C07261=1094.905,99.081,438.619,176.128,17.125,152.423
C07262=1094.899,98.832,438.636,176.125,17.124,152.424
C07263=1094.893,98.582,438.654,176.123,17.123,152.424
C07264=1094.888,98.333,438.673,176.120,17.123,152.424
C07265=1094.882,98.083,438.691,176.117,17.121,152.425
C07266=1094.877,97.834,438.709,176.115,17.121,152.425
C07267=1094.870,97.585,438.726,176.112,17.120,152.425
C07268=1094.865,97.336,438.745,176.110,17.119,152.426
C07269=1094.859,97.086,438.763,176.108,17.118,152.426
C07270=1094.854,96.837,438.781,176.106,17.117,152.426
C07271=1094.848,96.587,438.799,176.103,17.117,152.426
C07272=1094.843,96.339,438.818,176.100,17.115,152.427
C07273=1094.836,96.063,438.837,176.098,17.115,152.427
C07274=1094.830,95.788,438.857,176.095,17.114,152.427
C07275=1094.824,95.513,438.877,176.093,17.113,152.428
C07276=1094.817,95.237,438.896,176.090,17.112,152.428
C07277=1094.812,94.988,438.915,176.087,17.111,152.428
C07278=1094.806,94.739,438.933,176.085,17.110,152.429
C07279=1094.801,94.490,438.951,176.082,17.109,152.429
C07280=1094.794,94.240,438.969,176.080,17.108,152.429
C07281=1094.790,93.991,438.987,176.077,17.108,152.430
C07282=1094.784,93.741,439.005,176.075,17.107,152.430
C07283=1094.778,93.492,439.022,176.073,17.106,152.430
C07284=1094.772,93.243,439.040,176.070,17.104,152.430
C07285=1094.767,92.993,439.059,176.068,17.104,152.431
C07286=1094.761,92.744,439.077,176.065,17.103,152.431
C07287=1094.756,92.495,439.094,176.063,17.102,152.431
C07288=1094.750,92.245,439.112,176.061,17.101,152.432
C07289=1094.744,91.996,439.130,176.059,17.101,152.432
C07290=1094.739,91.747,439.148,176.056,17.099,152.432
C07291=1094.733,91.497,439.166,176.054,17.099,152.432
C07292=1094.728,91.248,439.184,176.051,17.097,152.433
C07293=1094.722,90.999,439.201,176.048,17.097,152.433
C07294=1094.716,90.749,439.219,176.046,17.096,152.433
C07295=1094.711,90.500,439.237,176.044,17.095,152.434
C07296=1094.705,90.251,439.254,176.042,17.094,152.434
C07297=1094.699,90.002,439.272,176.039,17.093,152.434
C07298=1094.693,89.753,439.290,176.037,17.093,152.434
C07299=1094.688,89.504,439.307,176.034,17.092,152.435
C07300=1094.682,89.254,439.325,176.032,17.091,152.435
C07301=1094.676,89.005,439.343,176.030,17.090,152.435
C07302=1094.670,88.755,439.361,176.027,17.088,152.436
C07303=1094.665,88.506,439.378,176.025,17.088,152.436
C07304=1094.659,88.257,439.396,176.022,17.087,152.436
C07305=1094.653,88.007,439.414,176.020,17.086,152.436
C07306=1094.647,87.758,439.431,176.017,17.085,152.437
C07307=1094.642,87.509,439.449,176.015,17.084,152.437
C07308=1094.636,87.260,439.466,176.013,17.083,152.437
C07309=1094.631,87.010,439.484,176.011,17.083,152.437
C07310=1094.625,86.761,439.501,176.008,17.081,152.438
C07311=1094.620,86.512,439.519,176.006,17.081,152.438
C07312=1094.613,86.262,439.537,176.004,17.079,152.438
C07313=1094.608,86.013,439.554,176.001,17.078,152.439
C07314=1094.602,85.764,439.572,175.999,17.078,152.439
C07315=1094.596,85.514,439.590,175.996,17.076,152.439
C07316=1094.591,85.264,439.607,175.994,17.076,152.439
C07317=1094.586,85.015,439.624,175.992,17.074,152.440
C07318=1094.580,84.766,439.642,175.990,17.074,152.440
C07319=1094.574,84.517,439.660,175.987,17.073,152.440
C07320=1094.568,84.268,439.677,175.985,17.072,152.440
C07321=1094.563,84.018,439.694,175.982,17.071,152.441
C07322=1094.558,83.769,439.712,175.981,17.070,152.441
C07323=1094.552,83.519,439.730,175.978,17.069,152.441
C07324=1094.546,83.270,439.747,175.976,17.068,152.441
C07325=1094.540,83.021,439.763,175.973,17.067,152.442
C07326=1094.535,82.772,439.781,175.970,17.066,152.442
C07327=1094.529,82.523,439.799,175.969,17.065,152.442
C07328=1094.523,82.273,439.817,175.966,17.064,152.442
C07329=1094.518,82.023,439.833,175.964,17.063,152.443
C07330=1094.512,81.774,439.851,175.961,17.062,152.443
C07331=1094.507,81.525,439.869,175.959,17.061,152.443
C07332=1094.501,81.276,439.885,175.957,17.060,152.443
C07333=1094.495,81.026,439.903,175.955,17.059,152.444
C07334=1094.489,80.777,439.920,175.952,17.058,152.444
C07335=1094.484,80.527,439.937,175.950,17.058,152.444
C07336=1094.478,80.278,439.955,175.947,17.056,152.445
C07337=1094.472,80.003,439.974,175.945,17.055,152.445
C07338=1094.466,79.728,439.993,175.943,17.054,152.445
C07339=1094.460,79.452,440.012,175.940,17.053,152.445
C07340=1094.454,79.177,440.031,175.937,17.052,152.446
C07341=1094.448,78.928,440.049,175.935,17.050,152.446
C07342=1094.443,78.678,440.066,175.933,17.050,152.446
C07343=1094.437,78.429,440.082,175.930,17.048,152.446
C07344=1094.431,78.180,440.100,175.928,17.048,152.447
C07345=1094.425,77.930,440.117,175.926,17.047,152.447
C07346=1094.420,77.681,440.135,175.924,17.046,152.447
C07347=1094.414,77.431,440.151,175.921,17.045,152.447
C07348=1094.408,77.182,440.169,175.919,17.044,152.448
C07349=1094.403,76.933,440.186,175.917,17.043,152.448
C07350=1094.397,76.684,440.202,175.915,17.042,152.448
C07351=1094.391,76.434,440.220,175.912,17.040,152.448
C07352=1094.385,76.185,440.237,175.910,17.040,152.448
C07353=1094.379,75.935,440.254,175.908,17.039,152.449
C07354=1094.374,75.686,440.271,175.906,17.038,152.449
C07355=1094.369,75.437,440.288,175.903,17.037,152.449
C07356=1094.363,75.188,440.305,175.901,17.036,152.450
C07357=1094.357,74.938,440.322,175.899,17.034,152.450
C07358=1094.352,74.689,440.339,175.897,17.034,152.450
C07359=1094.345,74.439,440.356,175.894,17.033,152.450
C07360=1094.340,74.190,440.374,175.892,17.032,152.450
C07361=1094.334,73.940,440.390,175.889,17.031,152.451
C07362=1094.329,73.691,440.407,175.888,17.030,152.451
C07363=1094.323,73.442,440.424,175.885,17.028,152.451
C07364=1094.318,73.192,440.441,175.883,17.028,152.451
C07365=1094.312,72.944,440.458,175.880,17.026,152.452
C07366=1094.306,72.694,440.475,175.879,17.026,152.452
C07367=1094.300,72.445,440.491,175.876,17.024,152.452
C07368=1094.295,72.196,440.509,175.874,17.023,152.452
C07369=1094.290,71.946,440.526,175.872,17.022,152.452
C07370=1094.283,71.696,440.542,175.870,17.022,152.453
C07371=1094.278,71.447,440.560,175.867,17.020,152.453
C07372=1094.272,71.197,440.576,175.865,17.019,152.453
C07373=1094.266,70.948,440.593,175.863,17.018,152.453
C07374=1094.261,70.699,440.610,175.861,17.017,152.453
C07375=1094.255,70.449,440.627,175.858,17.016,152.454
C07376=1094.250,70.200,440.644,175.856,17.015,152.454
C07377=1094.243,69.951,440.660,175.854,17.014,152.454
C07378=1094.238,69.701,440.677,175.852,17.013,152.454
C07379=1094.232,69.452,440.694,175.849,17.011,152.455
C07380=1094.227,69.202,440.710,175.847,17.011,152.455
C07381=1094.221,68.954,440.727,175.845,17.010,152.455
C07382=1094.216,68.704,440.744,175.843,17.008,152.455
C07383=1094.210,68.455,440.761,175.840,17.007,152.456
C07384=1094.204,68.205,440.777,175.838,17.007,152.456
C07385=1094.198,67.956,440.794,175.836,17.005,152.456
C07386=1094.193,67.707,440.811,175.834,17.004,152.456
C07387=1094.187,67.457,440.827,175.831,17.003,152.456
C07388=1094.182,67.208,440.844,175.830,17.002,152.457
C07389=1094.176,66.958,440.861,175.827,17.001,152.457
C07390=1094.170,66.709,440.877,175.825,17.000,152.457
C07391=1094.164,66.460,440.894,175.824,16.999,152.457
C07392=1094.158,66.211,440.911,175.821,16.998,152.457
C07393=1094.153,65.961,440.928,175.819,16.997,152.458
C07394=1094.147,65.711,440.944,175.817,16.995,152.458
C07395=1094.141,65.462,440.960,175.815,16.995,152.458
C07396=1094.136,65.212,440.977,175.812,16.993,152.458
C07397=1094.130,64.963,440.993,175.810,16.992,152.458
C07398=1094.125,64.714,441.011,175.808,16.991,152.459
C07399=1094.119,64.465,441.027,175.806,16.990,152.459
C07400=1094.113,64.215,441.043,175.803,16.989,152.459
C07401=1094.106,63.940,441.061,175.801,16.988,152.459
C07402=1094.100,63.664,441.079,175.799,16.987,152.460
C07403=1094.093,63.389,441.097,175.796,16.986,152.460
C07404=1094.087,63.113,441.115,175.794,16.984,152.460
C07405=1094.082,62.864,441.133,175.792,16.983,152.460
C07406=1094.076,62.615,441.149,175.789,16.982,152.461
C07407=1094.070,62.366,441.165,175.787,16.981,152.461
C07408=1094.064,62.116,441.182,175.785,16.980,152.461
C07409=1094.058,61.867,441.198,175.783,16.979,152.461
C07410=1094.053,61.617,441.215,175.781,16.978,152.461
C07411=1094.047,61.368,441.231,175.778,16.977,152.462
C07412=1094.041,61.119,441.247,175.777,16.976,152.462
C07413=1094.035,60.869,441.264,175.774,16.974,152.462
C07414=1094.029,60.620,441.280,175.772,16.974,152.462
C07415=1094.024,60.370,441.297,175.770,16.972,152.462
C07416=1094.018,60.121,441.313,175.768,16.971,152.463
C07417=1094.012,59.871,441.328,175.765,16.970,152.463
C07418=1094.006,59.622,441.345,175.763,16.969,152.463
C07419=1094.000,59.372,441.361,175.762,16.968,152.463
C07420=1093.995,59.123,441.378,175.759,16.967,152.463
C07421=1093.989,58.873,441.394,175.757,16.966,152.464
C07422=1093.983,58.624,441.410,175.755,16.964,152.464
C07423=1093.978,58.375,441.426,175.753,16.964,152.464
C07424=1093.972,58.126,441.442,175.750,16.962,152.464
C07425=1093.966,57.877,441.459,175.749,16.961,152.464
C07426=1093.960,57.627,441.475,175.746,16.960,152.464
C07427=1093.955,57.377,441.491,175.744,16.959,152.465
C07428=1093.949,57.128,441.507,175.742,16.958,152.465
C07429=1093.943,56.878,441.524,175.740,16.957,152.465
C07430=1093.937,56.629,441.540,175.738,16.956,152.465
C07431=1093.931,56.380,441.556,175.736,16.954,152.465
C07432=1093.926,56.131,441.572,175.734,16.954,152.466
C07433=1093.920,55.881,441.588,175.731,16.952,152.466
C07434=1093.915,55.631,441.604,175.729,16.951,152.466
C07435=1093.909,55.382,441.621,175.727,16.949,152.466
C07436=1093.903,55.133,441.637,175.725,16.949,152.466
C07437=1093.897,54.883,441.653,175.723,16.947,152.467
C07438=1093.892,54.633,441.669,175.721,16.946,152.467
C07439=1093.886,54.385,441.685,175.719,16.945,152.467
C07440=1093.880,54.135,441.701,175.717,16.944,152.467
C07441=1093.874,53.886,441.717,175.715,16.943,152.467
C07442=1093.869,53.636,441.733,175.712,16.941,152.467
C07443=1093.863,53.387,441.749,175.710,16.941,152.468
C07444=1093.857,53.137,441.766,175.708,16.939,152.468
C07445=1093.852,52.888,441.781,175.706,16.938,152.468
C07446=1093.846,52.638,441.797,175.704,16.937,152.468
C07447=1093.841,52.389,441.813,175.702,16.935,152.468
C07448=1093.835,52.139,441.829,175.700,16.935,152.468
C07449=1093.829,51.890,441.845,175.698,16.933,152.469
C07450=1093.824,51.641,441.861,175.696,16.932,152.469
C07451=1093.818,51.391,441.877,175.693,16.931,152.469
C07452=1093.812,51.142,441.893,175.692,16.930,152.469
C07453=1093.806,50.892,441.909,175.690,16.929,152.469
C07454=1093.801,50.643,441.924,175.687,16.927,152.469
C07455=1093.795,50.394,441.941,175.686,16.926,152.470
C07456=1093.789,50.144,441.957,175.683,16.925,152.470
C07457=1093.783,49.894,441.972,175.681,16.924,152.470
C07458=1093.778,49.646,441.988,175.679,16.922,152.470
C07459=1093.772,49.396,442.004,175.677,16.921,152.470
C07460=1093.766,49.147,442.020,175.676,16.920,152.470
C07461=1093.761,48.897,442.036,175.673,16.919,152.471
C07462=1093.755,48.648,442.052,175.671,16.918,152.471
C07463=1093.750,48.399,442.068,175.669,16.916,152.471
C07464=1093.744,48.149,442.083,175.667,16.915,152.471
C07465=1093.738,47.873,442.101,175.664,16.914,152.471
C07466=1093.732,47.598,442.118,175.663,16.913,152.471
C07467=1093.726,47.321,442.136,175.660,16.911,152.472
C07468=1093.720,47.046,442.154,175.658,16.910,152.472
C07469=1093.714,46.796,442.169,175.656,16.909,152.472
C07470=1093.708,46.548,442.185,175.654,16.907,152.472
C07471=1093.702,46.298,442.200,175.652,16.906,152.472
C07472=1093.696,46.048,442.216,175.649,16.905,152.472
C07473=1093.691,45.799,442.231,175.648,16.904,152.472
C07474=1093.685,45.550,442.248,175.646,16.902,152.473
C07475=1093.680,45.300,442.263,175.643,16.901,152.473
C07476=1093.674,45.051,442.279,175.642,16.900,152.473
C07477=1093.669,44.801,442.295,175.639,16.898,152.473
C07478=1093.663,44.551,442.310,175.638,16.897,152.473
C07479=1093.658,44.303,442.326,175.636,16.897,152.473
C07480=1093.652,44.053,442.342,175.633,16.895,152.474
C07481=1093.647,43.804,442.358,175.632,16.894,152.474
C07482=1093.641,43.554,442.373,175.629,16.892,152.474
C07483=1093.635,43.304,442.389,175.627,16.891,152.474
C07484=1093.629,43.055,442.404,175.626,16.890,152.474
C07485=1093.624,42.806,442.420,175.623,16.889,152.474
C07486=1093.618,42.556,442.435,175.622,16.887,152.474
C07487=1093.612,42.306,442.451,175.619,16.886,152.475
C07488=1093.607,42.057,442.466,175.617,16.885,152.475
C07489=1093.600,41.808,442.482,175.616,16.884,152.475
C07490=1093.595,41.558,442.498,175.613,16.882,152.475
C07491=1093.590,41.309,442.513,175.611,16.882,152.475
C07492=1093.584,41.059,442.528,175.609,16.880,152.475
C07493=1093.578,40.811,442.544,175.607,16.879,152.475
C07494=1093.572,40.561,442.559,175.606,16.878,152.476
C07495=1093.567,40.311,442.575,175.603,16.876,152.476
C07496=1093.561,40.062,442.591,175.601,16.875,152.476
C07497=1093.555,39.812,442.606,175.599,16.874,152.476
C07498=1093.549,39.562,442.621,175.597,16.872,152.476
C07499=1093.544,39.313,442.636,175.596,16.871,152.476
C07500=1093.538,39.064,442.653,175.593,16.870,152.477
C07501=1093.532,38.815,442.667,175.591,16.869,152.477
C07502=1093.527,38.565,442.683,175.589,16.867,152.477
C07503=1093.521,38.315,442.698,175.587,16.866,152.477
C07504=1093.516,38.066,442.714,175.586,16.865,152.477
C07505=1093.509,37.817,442.729,175.583,16.864,152.477
C07506=1093.504,37.567,442.744,175.582,16.863,152.477
C07507=1093.498,37.318,442.759,175.580,16.861,152.477
C07508=1093.492,37.068,442.775,175.577,16.860,152.478
C07509=1093.487,36.818,442.790,175.576,16.859,152.478
C07510=1093.481,36.569,442.806,175.573,16.857,152.478
C07511=1093.476,36.320,442.821,175.572,16.856,152.478
C07512=1093.469,36.071,442.836,175.570,16.855,152.478
C07513=1093.464,35.821,442.851,175.567,16.853,152.478
C07514=1093.459,35.571,442.866,175.566,16.853,152.479
C07515=1093.452,35.322,442.881,175.564,16.852,152.479
C07516=1093.447,35.072,442.897,175.562,16.850,152.479
C07517=1093.440,34.823,442.912,175.560,16.849,152.479
C07518=1093.435,34.573,442.928,175.557,16.847,152.479
C07519=1093.429,34.324,442.942,175.556,16.847,152.479
C07520=1093.423,34.074,442.958,175.554,16.845,152.479
C07521=1093.418,33.825,442.972,175.552,16.844,152.479
C07522=1093.412,33.576,442.988,175.550,16.843,152.480
C07523=1093.406,33.327,443.003,175.548,16.841,152.480
C07524=1093.400,33.077,443.018,175.546,16.840,152.480
C07525=1093.395,32.827,443.034,175.544,16.839,152.480
C07526=1093.389,32.578,443.048,175.542,16.838,152.480
C07527=1093.383,32.328,443.064,175.540,16.836,152.480
C07528=1093.378,32.079,443.078,175.538,16.835,152.480
C07529=1093.371,31.803,443.095,175.536,16.833,152.480
C07530=1093.365,31.528,443.112,175.534,16.832,152.481
C07531=1093.359,31.252,443.129,175.532,16.831,152.481
C07532=1093.352,30.977,443.145,175.529,16.829,152.481
C07533=1093.347,30.727,443.161,175.527,16.828,152.481
C07534=1093.341,30.478,443.175,175.526,16.827,152.481
C07535=1093.335,30.228,443.191,175.523,16.825,152.481
C07536=1093.330,29.979,443.205,175.522,16.824,152.481
C07537=1093.324,29.729,443.221,175.520,16.823,152.482
C07538=1093.318,29.480,443.235,175.518,16.821,152.482
C07539=1093.312,29.230,443.251,175.516,16.820,152.482
C07540=1093.307,28.981,443.266,175.515,16.819,152.482
C07541=1093.301,28.731,443.280,175.512,16.817,152.482
C07542=1093.296,28.481,443.295,175.511,16.816,152.482
C07543=1093.289,28.232,443.310,175.508,16.815,152.482
C07544=1093.284,27.983,443.325,175.506,16.814,152.482
C07545=1093.278,27.733,443.340,175.505,16.813,152.483
C07546=1093.272,27.484,443.355,175.502,16.811,152.483
C07547=1093.266,27.234,443.370,175.501,16.810,152.483
C07548=1093.261,26.985,443.385,175.499,16.809,152.483
C07549=1093.254,26.735,443.399,175.496,16.807,152.483
C07550=1093.249,26.485,443.414,175.495,16.806,152.483
C07551=1093.244,26.236,443.429,175.493,16.805,152.483
C07552=1093.237,25.987,443.444,175.491,16.803,152.483
C07553=1093.232,25.738,443.459,175.489,16.802,152.483
C07554=1093.226,25.488,443.474,175.487,16.801,152.484
C07555=1093.220,25.238,443.488,175.485,16.800,152.484
C07556=1093.215,24.988,443.503,175.483,16.799,152.484
C07557=1093.209,24.739,443.518,175.482,16.797,152.484
C07558=1093.203,24.490,443.533,175.479,16.796,152.484
C07559=1093.197,24.240,443.548,175.478,16.795,152.484
C07560=1093.191,23.990,443.562,175.476,16.793,152.484
C07561=1093.186,23.741,443.577,175.474,16.792,152.485
C07562=1093.180,23.492,443.591,175.472,16.791,152.485
C07563=1093.174,23.242,443.607,175.470,16.789,152.485
C07564=1093.169,22.993,443.621,175.468,16.788,152.485
C07565=1093.162,22.743,443.636,175.466,16.787,152.485
C07566=1093.157,22.494,443.651,175.465,16.786,152.485
C07567=1093.152,22.244,443.665,175.462,16.784,152.485
C07568=1093.145,21.995,443.680,175.461,16.783,152.485
C07569=1093.140,21.746,443.694,175.459,16.782,152.485
C07570=1093.134,21.495,443.709,175.457,16.780,152.485
C07571=1093.129,21.246,443.724,175.455,16.779,152.486
C07572=1093.123,20.997,443.738,175.453,16.778,152.486
C07573=1093.117,20.747,443.752,175.451,16.776,152.486
C07574=1093.112,20.498,443.768,175.449,16.775,152.486
C07575=1093.105,20.248,443.783,175.448,16.774,152.486
C07576=1093.100,19.998,443.796,175.446,16.772,152.486
C07577=1093.094,19.749,443.811,175.444,16.771,152.486
C07578=1093.088,19.500,443.826,175.442,16.770,152.486
C07579=1093.082,19.250,443.840,175.440,16.769,152.486
C07580=1093.077,19.001,443.855,175.438,16.767,152.487
C07581=1093.071,18.751,443.869,175.436,16.766,152.487
C07582=1093.065,18.502,443.884,175.435,16.765,152.487
C07583=1093.059,18.252,443.899,175.432,16.763,152.487
C07584=1093.053,18.002,443.913,175.430,16.762,152.487
C07585=1093.048,17.753,443.927,175.429,16.761,152.487
C07586=1093.042,17.503,443.941,175.427,16.759,152.487
C07587=1093.036,17.254,443.957,175.425,16.758,152.487
C07588=1093.031,17.004,443.970,175.423,16.757,152.487
C07589=1093.025,16.755,443.985,175.422,16.755,152.488
C07590=1093.019,16.505,443.999,175.419,16.754,152.488
C07591=1093.013,16.256,444.014,175.418,16.753,152.488
C07592=1093.007,16.006,444.028,175.416,16.751,152.488
C07593=1093.001,15.733,444.044,175.414,16.750,152.488
C07594=1092.995,15.458,444.060,175.412,16.749,152.488
C07595=1092.988,15.184,444.076,175.410,16.747,152.488
C07596=1092.982,14.909,444.091,175.407,16.745,152.488
C07597=1092.976,14.660,444.106,175.406,16.744,152.488
C07598=1092.971,14.410,444.120,175.404,16.743,152.489
C07599=1092.965,14.162,444.135,175.402,16.742,152.489
C07600=1092.959,13.912,444.149,175.400,16.740,152.489
C07601=1092.953,13.663,444.163,175.398,16.739,152.489
C07602=1092.947,13.412,444.177,175.397,16.738,152.489
C07603=1092.941,13.163,444.191,175.394,16.736,152.489
C07604=1092.936,12.914,444.206,175.393,16.735,152.489
C07605=1092.929,12.663,444.220,175.391,16.734,152.489
C07606=1092.924,12.415,444.235,175.389,16.733,152.489
C07607=1092.918,12.165,444.248,175.387,16.731,152.490
C07608=1092.913,11.915,444.262,175.385,16.730,152.490
C07609=1092.906,11.666,444.277,175.384,16.729,152.490
C07610=1092.901,11.416,444.291,175.381,16.727,152.490
C07611=1092.895,11.167,444.306,175.380,16.726,152.490
C07612=1092.889,10.917,444.320,175.378,16.725,152.490
C07613=1092.883,10.668,444.333,175.376,16.724,152.490
C07614=1092.877,10.419,444.348,175.374,16.722,152.490
C07615=1092.871,10.168,444.362,175.372,16.721,152.490
C07616=1092.865,9.919,444.376,175.371,16.720,152.491
C07617=1092.860,9.670,444.391,175.368,16.718,152.491
C07618=1092.854,9.420,444.404,175.367,16.717,152.491
C07619=1092.848,9.170,444.419,175.365,16.716,152.491
C07620=1092.842,8.921,444.433,175.364,16.715,152.491
C07621=1092.836,8.672,444.446,175.361,16.713,152.491
C07622=1092.831,8.422,444.460,175.360,16.712,152.491
C07623=1092.825,8.172,444.475,175.358,16.711,152.491
C07624=1092.819,7.923,444.489,175.356,16.710,152.491
C07625=1092.813,7.673,444.503,175.354,16.708,152.492
C07626=1092.808,7.424,444.517,175.352,16.707,152.492
C07627=1092.802,7.174,444.531,175.351,16.705,152.492
C07628=1092.796,6.925,444.546,175.348,16.703,152.492
C07629=1092.790,6.675,444.559,175.347,16.702,152.492
C07630=1092.784,6.426,444.573,175.345,16.701,152.492
C07631=1092.778,6.176,444.587,175.344,16.700,152.492
C07632=1092.773,5.926,444.601,175.341,16.698,152.492
C07633=1092.767,5.677,444.615,175.340,16.697,152.492
C07634=1092.761,5.427,444.629,175.338,16.696,152.492
C07635=1092.755,5.178,444.643,175.336,16.695,152.492
C07636=1092.749,4.928,444.657,175.334,16.693,152.493
C07637=1092.744,4.678,444.671,175.332,16.692,152.493
C07638=1092.738,4.429,444.685,175.331,16.691,152.493
C07639=1092.732,4.180,444.699,175.329,16.689,152.493
C07640=1092.726,3.931,444.712,175.327,16.688,152.493
C07641=1092.721,3.681,444.726,175.325,16.686,152.493
C07642=1092.715,3.431,444.741,175.324,16.685,152.493
C07643=1092.709,3.181,444.754,175.322,16.684,152.493
C07644=1092.704,2.931,444.768,175.320,16.682,152.493
C07645=1092.697,2.682,444.782,175.318,16.681,152.493
C07646=1092.692,2.433,444.795,175.316,16.680,152.493
C07647=1092.686,2.184,444.810,175.315,16.679,152.493
C07648=1092.681,1.934,444.824,175.313,16.677,152.494
C07649=1092.675,1.684,444.838,175.311,16.676,152.494
C07650=1092.668,1.435,444.851,175.309,16.675,152.494
C07651=1092.663,1.185,444.865,175.308,16.673,152.494
C07652=1092.658,0.935,444.879,175.305,16.672,152.494
C07653=1092.652,0.686,444.893,175.304,16.671,152.494
C07654=1092.646,0.437,444.906,175.302,16.669,152.494
C07655=1092.640,0.187,444.920,175.301,16.668,152.494
C07656=1092.635,-0.063,444.934,175.298,16.666,152.494
C07657=1092.628,-0.335,444.949,175.297,16.665,152.494
C07658=1092.622,-0.607,444.964,175.294,16.663,152.495
C07659=1092.616,-0.880,444.979,175.293,16.662,152.495
C07660=1092.610,-1.152,444.994,175.291,16.660,152.495
C07661=1092.604,-1.401,445.008,175.289,16.659,152.495
C07662=1092.598,-1.650,445.021,175.287,16.658,152.495
C07663=1092.593,-1.900,445.035,175.286,16.657,152.495
C07664=1092.587,-2.150,445.049,175.283,16.655,152.495
C07665=1092.581,-2.400,445.062,175.282,16.654,152.495
C07666=1092.575,-2.649,445.076,175.280,16.652,152.495
C07667=1092.570,-2.899,445.090,175.279,16.651,152.495
C07668=1092.564,-3.148,445.104,175.277,16.650,152.495
C07669=1092.558,-3.398,445.117,175.275,16.648,152.495
C07670=1092.552,-3.647,445.131,175.273,16.647,152.496
C07671=1092.546,-3.896,445.144,175.272,16.646,152.496
C07672=1092.541,-4.146,445.158,175.270,16.645,152.496
C07673=1092.535,-4.396,445.171,175.267,16.643,152.496
C07674=1092.529,-4.645,445.184,175.266,16.641,152.496
C07675=1092.523,-4.895,445.198,175.265,16.640,152.496
C07676=1092.518,-5.144,445.212,175.263,16.639,152.496
C07677=1092.511,-5.394,445.225,175.261,16.638,152.496
C07678=1092.505,-5.644,445.239,175.259,16.636,152.496
C07679=1092.499,-5.893,445.252,175.257,16.635,152.496
C07680=1092.494,-6.143,445.265,175.256,16.634,152.496
C07681=1092.488,-6.393,445.279,175.254,16.633,152.497
C07682=1092.482,-6.642,445.293,175.252,16.631,152.497
C07683=1092.476,-6.891,445.306,175.250,16.630,152.497
C07684=1092.471,-7.141,445.320,175.249,16.628,152.497
C07685=1092.464,-7.390,445.333,175.247,16.627,152.497
C07686=1092.459,-7.640,445.346,175.245,16.626,152.497
C07687=1092.453,-7.890,445.359,175.243,16.624,152.497
C07688=1092.447,-8.139,445.373,175.241,16.623,152.497
C07689=1092.441,-8.389,445.387,175.240,16.622,152.497
C07690=1092.436,-8.639,445.400,175.238,16.621,152.497
C07691=1092.430,-8.888,445.413,175.236,16.619,152.497
C07692=1092.424,-9.137,445.426,175.234,16.618,152.497
C07693=1092.418,-9.387,445.440,175.233,16.617,152.498
C07694=1092.412,-9.637,445.453,175.231,16.615,152.498
C07695=1092.407,-9.886,445.467,175.230,16.614,152.498
C07696=1092.400,-10.136,445.480,175.227,16.613,152.498
C07697=1092.395,-10.386,445.494,175.226,16.611,152.498
C07698=1092.389,-10.636,445.507,175.224,16.610,152.498
C07699=1092.383,-10.885,445.520,175.223,16.609,152.498
C07700=1092.378,-11.134,445.533,175.221,16.608,152.498
C07701=1092.372,-11.384,445.546,175.219,16.606,152.498
C07702=1092.366,-11.633,445.560,175.217,16.605,152.498
C07703=1092.360,-11.883,445.573,175.215,16.604,152.499
C07704=1092.355,-12.133,445.586,175.214,16.602,152.498
C07705=1092.349,-12.382,445.599,175.212,16.601,152.499
C07706=1092.342,-12.631,445.613,175.210,16.599,152.499
C07707=1092.337,-12.881,445.626,175.208,16.598,152.499
C07708=1092.331,-13.131,445.639,175.207,16.597,152.499
C07709=1092.325,-13.380,445.653,175.205,16.596,152.499
C07710=1092.320,-13.630,445.666,175.204,16.594,152.499
C07711=1092.313,-13.879,445.679,175.201,16.592,152.499
C07712=1092.308,-14.130,445.692,175.200,16.591,152.499
C07713=1092.302,-14.379,445.705,175.198,16.590,152.499
C07714=1092.296,-14.629,445.719,175.196,16.589,152.499
C07715=1092.291,-14.878,445.732,175.195,16.587,152.499
C07716=1092.284,-15.128,445.745,175.194,16.586,152.499
C07717=1092.279,-15.378,445.758,175.191,16.585,152.500
C07718=1092.273,-15.627,445.771,175.189,16.583,152.500
C07719=1092.267,-15.877,445.784,175.188,16.582,152.500
C07720=1092.261,-16.126,445.797,175.186,16.581,152.500
C07721=1092.255,-16.397,445.811,175.184,16.579,152.500
C07722=1092.249,-16.667,445.826,175.182,16.578,152.500
C07723=1092.243,-16.938,445.840,175.181,16.577,152.500
C07724=1092.236,-17.209,445.854,175.178,16.575,152.500
C07725=1092.230,-17.458,445.867,175.177,16.574,152.500
C07726=1092.224,-17.708,445.880,175.175,16.573,152.500
C07727=1092.218,-17.957,445.893,175.174,16.572,152.501
C07728=1092.212,-18.207,445.906,175.172,16.570,152.501
C07729=1092.206,-18.456,445.919,175.170,16.569,152.501
C07730=1092.201,-18.706,445.931,175.168,16.567,152.501
C07731=1092.195,-18.955,445.945,175.167,16.566,152.501
C07732=1092.189,-19.205,445.957,175.165,16.565,152.501
C07733=1092.183,-19.454,445.971,175.163,16.564,152.501
C07734=1092.177,-19.704,445.984,175.162,16.563,152.501
C07735=1092.172,-19.954,445.996,175.159,16.561,152.501
C07736=1092.165,-20.203,446.010,175.158,16.560,152.501
C07737=1092.159,-20.453,446.022,175.156,16.558,152.501
C07738=1092.153,-20.703,446.035,175.155,16.557,152.501
C07739=1092.148,-20.953,446.048,175.153,16.556,152.502
C07740=1092.142,-21.201,446.061,175.152,16.555,152.502
C07741=1092.137,-21.451,446.074,175.150,16.554,152.502
C07742=1092.131,-21.701,446.087,175.148,16.552,152.502
C07743=1092.124,-21.950,446.100,175.146,16.551,152.502
C07744=1092.118,-22.200,446.112,175.145,16.549,152.502
C07745=1092.113,-22.450,446.125,175.143,16.548,152.502
C07746=1092.107,-22.700,446.139,175.141,16.547,152.502
C07747=1092.102,-22.949,446.151,175.140,16.546,152.502
C07748=1092.096,-23.199,446.163,175.137,16.544,152.502
C07749=1092.090,-23.448,446.177,175.136,16.543,152.502
C07750=1092.084,-23.698,446.189,175.134,16.541,152.502
C07751=1092.078,-23.948,446.202,175.133,16.540,152.503
C07752=1092.072,-24.197,446.215,175.131,16.539,152.503
C07753=1092.066,-24.446,446.227,175.130,16.538,152.503
C07754=1092.061,-24.696,446.240,175.128,16.537,152.503
C07755=1092.055,-24.946,446.254,175.126,16.535,152.503
C07756=1092.049,-25.196,446.266,175.124,16.533,152.503
C07757=1092.043,-25.445,446.279,175.123,16.532,152.503
C07758=1092.037,-25.695,446.291,175.121,16.531,152.503
C07759=1092.032,-25.944,446.304,175.119,16.530,152.503
C07760=1092.026,-26.194,446.317,175.118,16.529,152.503
C07761=1092.020,-26.444,446.329,175.115,16.527,152.503
C07762=1092.014,-26.694,446.342,175.114,16.525,152.503
C07763=1092.008,-26.942,446.355,175.112,16.524,152.504
C07764=1092.002,-27.192,446.367,175.111,16.523,152.504
C07765=1091.996,-27.442,446.380,175.109,16.522,152.504
C07766=1091.991,-27.692,446.393,175.108,16.521,152.504
C07767=1091.984,-27.941,446.406,175.106,16.520,152.504
C07768=1091.978,-28.191,446.418,175.104,16.519,152.504
C07769=1091.973,-28.440,446.431,175.102,16.517,152.504
C07770=1091.967,-28.690,446.443,175.101,16.515,152.504
C07771=1091.961,-28.940,446.456,175.099,16.514,152.504
C07772=1091.955,-29.190,446.468,175.097,16.513,152.504
C07773=1091.949,-29.439,446.481,175.096,16.512,152.504
C07774=1091.943,-29.689,446.494,175.094,16.511,152.505
C07775=1091.938,-29.938,446.506,175.092,16.510,152.505
C07776=1091.931,-30.188,446.518,175.091,16.508,152.505
C07777=1091.925,-30.438,446.531,175.088,16.507,152.505
C07778=1091.919,-30.687,446.543,175.087,16.505,152.505
C07779=1091.914,-30.937,446.555,175.085,16.504,152.505
C07780=1091.908,-31.186,446.569,175.084,16.503,152.505
C07781=1091.902,-31.436,446.581,175.082,16.502,152.505
C07782=1091.896,-31.686,446.594,175.081,16.501,152.505
C07783=1091.890,-31.935,446.606,175.079,16.499,152.505
C07784=1091.885,-32.185,446.619,175.077,16.498,152.505
C07785=1091.878,-32.455,446.632,175.075,16.497,152.506
C07786=1091.872,-32.724,446.646,175.074,16.495,152.506
C07787=1091.866,-32.994,446.659,175.072,16.494,152.506
C07788=1091.859,-33.264,446.672,175.070,16.493,152.506
C07789=1091.853,-33.513,446.684,175.068,16.491,152.506
C07790=1091.847,-33.763,446.697,175.066,16.490,152.506
C07791=1091.842,-34.013,446.709,175.065,16.489,152.506
C07792=1091.836,-34.262,446.722,175.063,16.488,152.506
C07793=1091.830,-34.512,446.734,175.062,16.487,152.506
C07794=1091.825,-34.761,446.746,175.060,16.485,152.506
C07795=1091.818,-35.010,446.759,175.059,16.484,152.506
C07796=1091.812,-35.260,446.772,175.057,16.483,152.506
C07797=1091.806,-35.511,446.783,175.055,16.481,152.507
C07798=1091.801,-35.760,446.796,175.053,16.480,152.507
C07799=1091.795,-36.010,446.808,175.051,16.479,152.507
C07800=1091.789,-36.260,446.821,175.050,16.477,152.507
C07801=1091.783,-36.509,446.832,175.048,16.476,152.507
C07802=1091.777,-36.759,446.845,175.047,16.475,152.507
C07803=1091.771,-37.008,446.857,175.045,16.474,152.507
C07804=1091.766,-37.258,446.870,175.044,16.472,152.507
C07805=1091.760,-37.507,446.882,175.042,16.471,152.507
C07806=1091.754,-37.757,446.895,175.040,16.470,152.507
C07807=1091.748,-38.006,446.906,175.039,16.469,152.507
C07808=1091.742,-38.256,446.919,175.037,16.468,152.508
C07809=1091.736,-38.506,446.931,175.035,16.466,152.508
C07810=1091.731,-38.755,446.944,175.033,16.465,152.508
C07811=1091.724,-39.005,446.955,175.032,16.463,152.508
C07812=1091.718,-39.255,446.968,175.030,16.462,152.508
C07813=1091.713,-39.504,446.980,175.029,16.461,152.508
C07814=1091.707,-39.754,446.991,175.027,16.460,152.508
C07815=1091.701,-40.004,447.004,175.025,16.459,152.508
C07816=1091.695,-40.253,447.016,175.024,16.458,152.508
C07817=1091.689,-40.503,447.028,175.022,16.457,152.508
C07818=1091.683,-40.753,447.041,175.020,16.456,152.508
C07819=1091.677,-41.002,447.053,175.019,16.454,152.509
C07820=1091.671,-41.252,447.064,175.017,16.453,152.509
C07821=1091.665,-41.502,447.077,175.016,16.452,152.509
C07822=1091.659,-41.751,447.089,175.013,16.450,152.509
C07823=1091.653,-42.001,447.101,175.012,16.449,152.509
C07824=1091.648,-42.250,447.113,175.010,16.448,152.509
C07825=1091.641,-42.499,447.125,175.009,16.446,152.509
C07826=1091.636,-42.750,447.137,175.007,16.445,152.509
C07827=1091.629,-42.999,447.149,175.005,16.444,152.509
C07828=1091.624,-43.249,447.161,175.004,16.443,152.509
C07829=1091.618,-43.498,447.174,175.002,16.442,152.510
C07830=1091.612,-43.749,447.185,175.001,16.441,152.510
C07831=1091.606,-43.998,447.197,174.999,16.440,152.510
C07832=1091.600,-44.247,447.209,174.997,16.439,152.510
C07833=1091.594,-44.497,447.221,174.996,16.437,152.510
C07834=1091.589,-44.747,447.233,174.994,16.436,152.510
C07835=1091.582,-44.997,447.245,174.992,16.435,152.510
C07836=1091.577,-45.246,447.257,174.991,16.434,152.510
C07837=1091.570,-45.495,447.269,174.990,16.432,152.510
C07838=1091.565,-45.746,447.281,174.988,16.431,152.510
C07839=1091.559,-45.995,447.293,174.985,16.430,152.510
C07840=1091.553,-46.245,447.305,174.984,16.428,152.511
C07841=1091.548,-46.494,447.317,174.982,16.427,152.511
C07842=1091.541,-46.744,447.328,174.981,16.426,152.511
C07843=1091.536,-46.993,447.341,174.979,16.425,152.511
C07844=1091.529,-47.243,447.352,174.977,16.424,152.511
C07845=1091.523,-47.493,447.364,174.976,16.423,152.511
C07846=1091.517,-47.742,447.376,174.974,16.422,152.511
C07847=1091.512,-47.993,447.388,174.973,16.420,152.511
C07848=1091.506,-48.242,447.400,174.971,16.419,152.511
C07849=1091.500,-48.512,447.413,174.969,16.418,152.511
C07850=1091.493,-48.782,447.425,174.968,16.417,152.512
C07851=1091.487,-49.052,447.438,174.966,16.415,152.512
C07852=1091.480,-49.322,447.451,174.964,16.414,152.512
C07853=1091.475,-49.572,447.463,174.962,16.413,152.512
C07854=1091.469,-49.821,447.475,174.961,16.411,152.512
C07855=1091.463,-50.071,447.487,174.959,16.410,152.512
C07856=1091.457,-50.320,447.498,174.958,16.409,152.512
C07857=1091.451,-50.570,447.511,174.956,16.408,152.512
C07858=1091.445,-50.820,447.521,174.954,16.407,152.512
C07859=1091.439,-51.070,447.534,174.953,16.406,152.512
C07860=1091.433,-51.320,447.545,174.951,16.405,152.513
C07861=1091.427,-51.569,447.557,174.949,16.404,152.513
C07862=1091.420,-51.818,447.569,174.948,16.402,152.513
C07863=1091.415,-52.068,447.580,174.946,16.401,152.513
C07864=1091.409,-52.318,447.592,174.945,16.400,152.513
C07865=1091.402,-52.568,447.603,174.943,16.399,152.513
C07866=1091.397,-52.817,447.616,174.941,16.398,152.513
C07867=1091.391,-53.067,447.627,174.940,16.397,152.513
C07868=1091.385,-53.316,447.639,174.938,16.396,152.514
C07869=1091.378,-53.566,447.650,174.936,16.395,152.514
C07870=1091.373,-53.816,447.662,174.935,16.394,152.514
C07871=1091.367,-54.066,447.673,174.933,16.393,152.514
C07872=1091.360,-54.315,447.685,174.931,16.392,152.514
C07873=1091.355,-54.565,447.697,174.930,16.390,152.514
C07874=1091.348,-54.815,447.709,174.928,16.389,152.514
C07875=1091.343,-55.064,447.719,174.927,16.388,152.514
C07876=1091.336,-55.314,447.731,174.925,16.387,152.514
C07877=1091.331,-55.564,447.743,174.923,16.386,152.514
C07878=1091.324,-55.813,447.755,174.922,16.385,152.515
C07879=1091.319,-56.063,447.766,174.920,16.384,152.515
C07880=1091.312,-56.313,447.777,174.918,16.382,152.515
C07881=1091.307,-56.562,447.789,174.917,16.381,152.515
C07882=1091.301,-56.812,447.800,174.915,16.380,152.515
C07883=1091.295,-57.061,447.812,174.914,16.379,152.515
C07884=1091.288,-57.311,447.823,174.912,16.378,152.515
C07885=1091.282,-57.560,447.835,174.910,16.377,152.515
C07886=1091.277,-57.811,447.847,174.909,16.376,152.515
C07887=1091.271,-58.060,447.858,174.907,16.375,152.516
C07888=1091.264,-58.310,447.870,174.905,16.374,152.516
C07889=1091.259,-58.559,447.880,174.904,16.373,152.516
C07890=1091.253,-58.810,447.892,174.902,16.372,152.516
C07891=1091.247,-59.058,447.904,174.900,16.370,152.516
C07892=1091.241,-59.309,447.915,174.899,16.369,152.516
C07893=1091.235,-59.558,447.927,174.897,16.368,152.516
C07894=1091.228,-59.808,447.938,174.896,16.367,152.516
C07895=1091.223,-60.058,447.949,174.894,16.366,152.517
C07896=1091.217,-60.307,447.961,174.892,16.365,152.517
C07897=1091.211,-60.557,447.972,174.891,16.364,152.517
C07898=1091.204,-60.807,447.983,174.889,16.363,152.517
C07899=1091.198,-61.056,447.995,174.888,16.361,152.517
C07900=1091.193,-61.305,448.006,174.886,16.360,152.517
C07901=1091.187,-61.556,448.018,174.884,16.359,152.517
C07902=1091.181,-61.805,448.029,174.883,16.358,152.517
C07903=1091.175,-62.055,448.041,174.881,16.357,152.517
C07904=1091.169,-62.304,448.051,174.879,16.356,152.518
C07905=1091.163,-62.554,448.063,174.878,16.355,152.518
C07906=1091.157,-62.804,448.074,174.876,16.354,152.518
C07907=1091.152,-63.053,448.086,174.874,16.353,152.518
C07908=1091.145,-63.303,448.097,174.873,16.352,152.518
C07909=1091.139,-63.553,448.108,174.872,16.351,152.518
C07910=1091.133,-63.803,448.119,174.870,16.350,152.518
C07911=1091.127,-64.052,448.131,174.869,16.349,152.518
C07912=1091.121,-64.301,448.142,174.867,16.348,152.518
C07913=1091.115,-64.574,448.154,174.865,16.347,152.519
C07914=1091.109,-64.844,448.167,174.863,16.345,152.519
C07915=1091.102,-65.116,448.178,174.861,16.344,152.519
C07916=1091.096,-65.387,448.191,174.860,16.343,152.519
C07917=1091.089,-65.637,448.202,174.858,16.342,152.519
C07918=1091.084,-65.886,448.213,174.856,16.341,152.519
C07919=1091.078,-66.136,448.224,174.855,16.340,152.519
C07920=1091.072,-66.386,448.236,174.853,16.339,152.519
C07921=1091.066,-66.635,448.247,174.851,16.337,152.520
C07922=1091.060,-66.885,448.258,174.851,16.337,152.520
C07923=1091.054,-67.135,448.269,174.849,16.336,152.520
C07924=1091.048,-67.384,448.280,174.847,16.335,152.520
C07925=1091.043,-67.634,448.291,174.846,16.334,152.520
C07926=1091.036,-67.884,448.302,174.844,16.332,152.520
C07927=1091.031,-68.134,448.313,174.843,16.331,152.520
C07928=1091.025,-68.383,448.324,174.841,16.330,152.520
C07929=1091.019,-68.633,448.337,174.839,16.329,152.521
C07930=1091.013,-68.883,448.348,174.837,16.328,152.521
C07931=1091.007,-69.132,448.358,174.836,16.327,152.521
C07932=1091.001,-69.382,448.370,174.834,16.326,152.521
C07933=1090.995,-69.632,448.381,174.833,16.325,152.521
C07934=1090.990,-69.881,448.391,174.831,16.324,152.521
C07935=1090.983,-70.131,448.403,174.829,16.323,152.521
C07936=1090.978,-70.381,448.414,174.828,16.322,152.521
C07937=1090.972,-70.630,448.424,174.826,16.320,152.521
C07938=1090.966,-70.880,448.435,174.825,16.320,152.521
C07939=1090.960,-71.130,448.447,174.823,16.319,152.522
C07940=1090.954,-71.380,448.457,174.822,16.318,152.522
C07941=1090.948,-71.629,448.468,174.820,16.317,152.522
C07942=1090.942,-71.879,448.480,174.819,16.316,152.522
C07943=1090.936,-72.129,448.490,174.817,16.315,152.522
C07944=1090.931,-72.378,448.502,174.815,16.314,152.522
C07945=1090.925,-72.628,448.513,174.814,16.312,152.522
C07946=1090.919,-72.878,448.524,174.812,16.311,152.522
C07947=1090.913,-73.128,448.535,174.810,16.311,152.523
C07948=1090.908,-73.377,448.546,174.809,16.310,152.523
C07949=1090.902,-73.627,448.557,174.807,16.308,152.523
C07950=1090.896,-73.877,448.568,174.806,16.308,152.523
C07951=1090.890,-74.126,448.579,174.805,16.307,152.523
C07952=1090.884,-74.376,448.590,174.803,16.306,152.523
C07953=1090.878,-74.625,448.600,174.801,16.304,152.523
C07954=1090.871,-74.875,448.611,174.799,16.304,152.524
C07955=1090.865,-75.125,448.622,174.798,16.303,152.524
C07956=1090.860,-75.374,448.633,174.796,16.302,152.524
C07957=1090.853,-75.624,448.644,174.795,16.300,152.524
C07958=1090.848,-75.874,448.655,174.793,16.299,152.524
C07959=1090.842,-76.123,448.666,174.791,16.299,152.524
C07960=1090.835,-76.373,448.676,174.790,16.298,152.524
C07961=1090.829,-76.623,448.687,174.789,16.297,152.524
C07962=1090.824,-76.873,448.698,174.787,16.296,152.525
C07963=1090.818,-77.122,448.708,174.785,16.295,152.525
C07964=1090.812,-77.373,448.720,174.783,16.294,152.525
C07965=1090.806,-77.622,448.731,174.782,16.293,152.525
C07966=1090.799,-77.871,448.741,174.780,16.292,152.525
C07967=1090.794,-78.121,448.752,174.779,16.291,152.525
C07968=1090.787,-78.371,448.763,174.777,16.290,152.526
C07969=1090.782,-78.621,448.773,174.776,16.289,152.526
C07970=1090.776,-78.870,448.784,174.774,16.288,152.526
C07971=1090.770,-79.120,448.795,174.773,16.287,152.526
C07972=1090.764,-79.369,448.805,174.771,16.287,152.526
C07973=1090.758,-79.619,448.816,174.769,16.285,152.526
C07974=1090.752,-79.869,448.827,174.768,16.284,152.526
C07975=1090.746,-80.119,448.837,174.766,16.283,152.526
C07976=1090.740,-80.368,448.848,174.765,16.283,152.527
C07977=1090.734,-80.642,448.860,174.762,16.281,152.527
C07978=1090.727,-80.915,448.872,174.761,16.280,152.527
C07979=1090.721,-81.189,448.883,174.759,16.280,152.527
C07980=1090.714,-81.463,448.895,174.757,16.278,152.527
C07981=1090.707,-81.713,448.906,174.756,16.277,152.527
C07982=1090.701,-81.962,448.916,174.755,16.277,152.528
C07983=1090.695,-82.211,448.927,174.753,16.276,152.528
C07984=1090.689,-82.461,448.937,174.751,16.275,152.528
C07985=1090.682,-82.711,448.948,174.749,16.274,152.528
C07986=1090.677,-82.961,448.959,174.748,16.273,152.528
C07987=1090.670,-83.210,448.969,174.746,16.272,152.528
C07988=1090.665,-83.460,448.979,174.745,16.272,152.528
C07989=1090.658,-83.710,448.991,174.743,16.271,152.529
C07990=1090.652,-83.960,449.001,174.742,16.270,152.529
C07991=1090.647,-84.210,449.011,174.740,16.269,152.529
C07992=1090.640,-84.459,449.021,174.738,16.268,152.529
C07993=1090.634,-84.708,449.032,174.736,16.267,152.529
C07994=1090.628,-84.958,449.043,174.735,16.266,152.529
C07995=1090.622,-85.208,449.053,174.734,16.266,152.529
C07996=1090.616,-85.458,449.064,174.732,16.265,152.530
C07997=1090.610,-85.707,449.074,174.730,16.264,152.530
C07998=1090.604,-85.957,449.084,174.729,16.263,152.530
C07999=1090.598,-86.207,449.096,174.727,16.262,152.530
C08000=1090.591,-86.456,449.106,174.725,16.261,152.530
C08001=1090.586,-86.707,449.116,174.725,16.260,152.530
C08002=1090.579,-86.956,449.126,174.723,16.260,152.531
C08003=1090.574,-87.205,449.137,174.721,16.259,152.531
C08004=1090.568,-87.456,449.148,174.719,16.258,152.531
C08005=1090.561,-87.705,449.158,174.717,16.257,152.531
C08006=1090.555,-87.955,449.169,174.717,16.256,152.531
C08007=1090.549,-88.204,449.178,174.715,16.256,152.531
C08008=1090.544,-88.454,449.189,174.713,16.255,152.532
C08009=1090.537,-88.704,449.199,174.712,16.253,152.532
C08010=1090.531,-88.954,449.210,174.710,16.253,152.532
C08011=1090.525,-89.203,449.221,174.708,16.252,152.532
C08012=1090.519,-89.453,449.231,174.707,16.251,152.532
C08013=1090.513,-89.703,449.241,174.705,16.251,152.532
C08014=1090.507,-89.953,449.251,174.704,16.249,152.533
C08015=1090.501,-90.202,449.262,174.702,16.249,152.533
C08016=1090.495,-90.452,449.271,174.700,16.248,152.533
C08017=1090.490,-90.701,449.282,174.699,16.247,152.533
C08018=1090.482,-90.951,449.293,174.697,16.246,152.533
C08019=1090.477,-91.201,449.303,174.696,16.245,152.533
C08020=1090.471,-91.450,449.313,174.694,16.245,152.534
C08021=1090.465,-91.701,449.324,174.692,16.244,152.534
C08022=1090.459,-91.950,449.334,174.691,16.242,152.534
C08023=1090.453,-92.200,449.344,174.690,16.242,152.534
C08024=1090.447,-92.449,449.355,174.688,16.241,152.534
C08025=1090.441,-92.699,449.364,174.686,16.241,152.534
C08026=1090.436,-92.949,449.375,174.684,16.239,152.535
C08027=1090.429,-93.199,449.385,174.683,16.238,152.535
C08028=1090.423,-93.449,449.396,174.682,16.238,152.535
C08029=1090.417,-93.698,449.406,174.680,16.237,152.535
C08030=1090.411,-93.948,449.417,174.678,16.237,152.535
C08031=1090.405,-94.198,449.426,174.677,16.235,152.535
C08032=1090.399,-94.447,449.437,174.675,16.235,152.536
C08033=1090.393,-94.697,449.447,174.674,16.234,152.536
C08034=1090.388,-94.947,449.457,174.672,16.233,152.536
C08035=1090.381,-95.196,449.467,174.670,16.232,152.536
C08036=1090.376,-95.446,449.477,174.669,16.231,152.536
C08037=1090.369,-95.696,449.487,174.668,16.231,152.536
C08038=1090.364,-95.946,449.498,174.666,16.230,152.536
C08039=1090.357,-96.195,449.508,174.664,16.230,152.537
C08040=1090.351,-96.445,449.517,174.663,16.228,152.537
C08041=1090.344,-96.721,449.529,174.661,16.228,152.537
C08042=1090.338,-96.997,449.540,174.659,16.227,152.537
C08043=1090.332,-97.272,449.551,174.657,16.226,152.537
C08044=1090.325,-97.548,449.563,174.655,16.225,152.538
C08045=1090.319,-97.798,449.572,174.654,16.225,152.538
C08046=1090.313,-98.048,449.583,174.653,16.224,152.538
C08047=1090.307,-98.297,449.593,174.651,16.223,152.538
C08048=1090.301,-98.547,449.602,174.649,16.222,152.538
C08049=1090.295,-98.797,449.613,174.648,16.222,152.539
C08050=1090.289,-99.047,449.623,174.646,16.221,152.539
C08051=1090.282,-99.296,449.632,174.645,16.220,152.539
C08052=1090.277,-99.546,449.643,174.643,16.219,152.539
C08053=1090.271,-99.796,449.653,174.642,16.219,152.539
C08054=1090.264,-100.045,449.662,174.640,16.218,152.539
C08055=1090.258,-100.295,449.673,174.638,16.217,152.540
C08056=1090.252,-100.545,449.683,174.636,16.217,152.540
C08057=1090.246,-100.795,449.693,174.636,16.216,152.540
C08058=1090.239,-101.044,449.703,174.634,16.215,152.540
C08059=1090.234,-101.295,449.713,174.632,16.214,152.540
C08060=1090.228,-101.544,449.723,174.630,16.214,152.541
C08061=1090.221,-101.793,449.733,174.629,16.213,152.541
C08062=1090.215,-102.043,449.743,174.627,16.212,152.541
C08063=1090.210,-102.293,449.753,174.626,16.212,152.541
C08064=1090.203,-102.543,449.762,174.624,16.211,152.541
C08065=1090.197,-102.792,449.773,174.623,16.211,152.541
C08066=1090.191,-103.042,449.782,174.621,16.209,152.542
C08067=1090.185,-103.292,449.792,174.619,16.209,152.542
C08068=1090.179,-103.542,449.802,174.617,16.208,152.542
C08069=1090.173,-103.791,449.812,174.617,16.208,152.542
C08070=1090.166,-104.041,449.822,174.615,16.207,152.542
C08071=1090.161,-104.291,449.832,174.613,16.206,152.543
C08072=1090.155,-104.541,449.842,174.611,16.205,152.543
C08073=1090.148,-104.790,449.852,174.610,16.205,152.543
C08074=1090.142,-105.040,449.861,174.608,16.204,152.543
C08075=1090.137,-105.290,449.872,174.607,16.203,152.543
C08076=1090.131,-105.540,449.881,174.606,16.203,152.543
C08077=1090.124,-105.790,449.891,174.604,16.202,152.544
C08078=1090.118,-106.039,449.901,174.602,16.202,152.544
C08079=1090.112,-106.289,449.911,174.600,16.200,152.544
C08080=1090.106,-106.539,449.921,174.599,16.200,152.544
C08081=1090.100,-106.789,449.930,174.597,16.200,152.545
C08082=1090.094,-107.038,449.940,174.596,16.199,152.545
C08083=1090.088,-107.288,449.949,174.595,16.199,152.545
C08084=1090.081,-107.537,449.960,174.593,16.197,152.545
C08085=1090.075,-107.787,449.969,174.591,16.197,152.545
C08086=1090.070,-108.037,449.979,174.589,16.196,152.546
C08087=1090.064,-108.286,449.989,174.588,16.196,152.546
C08088=1090.058,-108.536,449.998,174.586,16.195,152.546
C08089=1090.052,-108.786,450.008,174.585,16.194,152.546
C08090=1090.046,-109.036,450.017,174.583,16.194,152.546
C08091=1090.039,-109.285,450.028,174.582,16.193,152.547
C08092=1090.033,-109.535,450.037,174.580,16.193,152.547
C08093=1090.027,-109.784,450.047,174.579,16.193,152.547
C08094=1090.021,-110.034,450.056,174.577,16.191,152.547
C08095=1090.015,-110.284,450.066,174.575,16.191,152.547
C08096=1090.008,-110.534,450.075,174.573,16.190,152.548
C08097=1090.002,-110.784,450.085,174.572,16.190,152.548
C08098=1089.997,-111.034,450.095,174.571,16.189,152.548
C08099=1089.991,-111.284,450.105,174.569,16.188,152.548
C08100=1089.984,-111.533,450.114,174.568,16.188,152.548
C08101=1089.978,-111.783,450.124,174.566,16.187,152.549
C08102=1089.972,-112.033,450.133,174.564,16.187,152.549
C08103=1089.966,-112.282,450.144,174.563,16.187,152.549
C08104=1089.959,-112.532,450.153,174.561,16.186,152.549
C08105=1089.953,-112.801,450.163,174.559,16.185,152.549
C08106=1089.947,-113.071,450.173,174.558,16.184,152.550
C08107=1089.940,-113.340,450.184,174.556,16.184,152.550
C08108=1089.934,-113.609,450.194,174.555,16.183,152.550
C08109=1089.927,-113.859,450.203,174.553,16.183,152.550
C08110=1089.921,-114.109,450.213,174.551,16.182,152.551
C08111=1089.915,-114.358,450.222,174.550,16.182,152.551
C08112=1089.909,-114.608,450.232,174.548,16.181,152.551
C08113=1089.903,-114.858,450.242,174.546,16.180,152.551
C08114=1089.896,-115.108,450.251,174.545,16.180,152.551
C08115=1089.890,-115.358,450.261,174.543,16.179,152.552
C08116=1089.884,-115.607,450.270,174.541,16.179,152.552
C08117=1089.879,-115.857,450.279,174.540,16.179,152.552
C08118=1089.872,-116.106,450.289,174.538,16.178,152.552
C08119=1089.866,-116.356,450.299,174.537,16.177,152.553
C08120=1089.860,-116.606,450.308,174.536,16.177,152.553
C08121=1089.854,-116.856,450.318,174.534,16.176,152.553
C08122=1089.848,-117.106,450.327,174.532,16.175,152.553
C08123=1089.842,-117.355,450.337,174.531,16.175,152.553
C08124=1089.835,-117.605,450.346,174.529,16.175,152.554
C08125=1089.829,-117.855,450.356,174.527,16.174,152.554
C08126=1089.824,-118.104,450.365,174.526,16.174,152.554
C08127=1089.817,-118.354,450.374,174.524,16.173,152.554
C08128=1089.811,-118.604,450.383,174.523,16.173,152.555
C08129=1089.805,-118.854,450.393,174.521,16.172,152.555
C08130=1089.799,-119.104,450.402,174.519,16.172,152.555
C08131=1089.792,-119.353,450.412,174.518,16.172,152.555
C08132=1089.786,-119.603,450.421,174.517,16.171,152.555
C08133=1089.780,-119.853,450.431,174.515,16.170,152.556
C08134=1089.774,-120.102,450.440,174.514,16.170,152.556
C08135=1089.768,-120.352,450.450,174.512,16.169,152.556
C08136=1089.762,-120.602,450.458,174.510,16.169,152.556
C08137=1089.755,-120.852,450.467,174.509,16.169,152.557
C08138=1089.749,-121.102,450.477,174.507,16.168,152.557
C08139=1089.743,-121.351,450.487,174.506,16.168,152.557
C08140=1089.737,-121.601,450.496,174.504,16.167,152.557
C08141=1089.731,-121.850,450.505,174.502,16.166,152.558
C08142=1089.726,-122.101,450.514,174.501,16.166,152.558
C08143=1089.719,-122.350,450.523,174.499,16.165,152.558
C08144=1089.712,-122.600,450.533,174.497,16.165,152.558
C08145=1089.706,-122.850,450.542,174.496,16.165,152.559
C08146=1089.700,-123.100,450.552,174.494,16.164,152.559
C08147=1089.695,-123.349,450.560,174.493,16.164,152.559
C08148=1089.689,-123.599,450.570,174.491,16.163,152.559
C08149=1089.682,-123.849,450.579,174.489,16.163,152.560
C08150=1089.676,-124.098,450.588,174.488,16.163,152.560
C08151=1089.669,-124.348,450.598,174.487,16.162,152.560
C08152=1089.664,-124.598,450.607,174.485,16.161,152.560
C08153=1089.658,-124.848,450.616,174.484,16.161,152.560
C08154=1089.651,-125.097,450.625,174.482,16.160,152.561
C08155=1089.645,-125.347,450.635,174.480,16.160,152.561
C08156=1089.639,-125.597,450.643,174.479,16.160,152.561
C08157=1089.633,-125.847,450.653,174.477,16.159,152.561
C08158=1089.627,-126.096,450.662,174.476,16.159,152.562
C08159=1089.620,-126.346,450.671,174.474,16.158,152.562
C08160=1089.615,-126.596,450.680,174.473,16.158,152.562
C08161=1089.608,-126.846,450.689,174.471,16.158,152.562
C08162=1089.601,-127.095,450.699,174.469,16.157,152.563
C08163=1089.596,-127.346,450.707,174.468,16.157,152.563
C08164=1089.590,-127.595,450.717,174.466,16.156,152.563
C08165=1089.583,-127.853,450.726,174.465,16.156,152.563
C08166=1089.577,-128.112,450.736,174.463,16.156,152.564
C08167=1089.576,-128.370,450.746,174.461,16.154,152.564
C08168=1089.582,-128.625,450.760,174.461,16.150,152.563
C08169=1089.177,-128.647,450.637,174.420,16.256,152.591
C08170=1089.171,-128.391,450.624,174.420,16.259,152.592
C08171=1089.171,-128.133,450.613,174.421,16.261,152.592
C08172=1089.177,-127.875,450.603,174.423,16.262,152.592
C08173=1089.184,-127.617,450.594,174.424,16.262,152.592
C08174=1089.190,-127.367,450.585,174.426,16.262,152.591
C08175=1089.196,-127.117,450.575,174.427,16.262,152.591
C08176=1089.202,-126.868,450.567,174.429,16.263,152.591
C08177=1089.208,-126.618,450.558,174.431,16.264,152.591
C08178=1089.215,-126.368,450.548,174.432,16.264,152.590
C08179=1089.221,-126.118,450.539,174.434,16.264,152.590
C08180=1089.228,-125.869,450.530,174.435,16.265,152.590
C08181=1089.233,-125.618,450.521,174.437,16.266,152.590
C08182=1089.239,-125.369,450.512,174.439,16.266,152.590
C08183=1089.246,-125.120,450.503,174.440,16.266,152.589
C08184=1089.252,-124.870,450.493,174.442,16.267,152.589
C08185=1089.258,-124.620,450.484,174.443,16.267,152.589
C08186=1089.264,-124.370,450.475,174.445,16.267,152.589
C08187=1089.270,-124.121,450.466,174.447,16.268,152.588
C08188=1089.277,-123.871,450.457,174.448,16.268,152.588
C08189=1089.283,-123.621,450.448,174.450,16.269,152.588
C08190=1089.289,-123.371,450.438,174.451,16.269,152.588
C08191=1089.295,-123.121,450.429,174.452,16.270,152.588
C08192=1089.301,-122.871,450.419,174.454,16.271,152.587
C08193=1089.307,-122.622,450.410,174.455,16.271,152.587
C08194=1089.313,-122.372,450.402,174.457,16.271,152.587
C08195=1089.319,-122.122,450.392,174.459,16.272,152.586
C08196=1089.326,-121.873,450.383,174.460,16.272,152.586
C08197=1089.332,-121.623,450.373,174.462,16.272,152.586
C08198=1089.338,-121.373,450.363,174.464,16.274,152.586
C08199=1089.343,-121.124,450.354,174.465,16.274,152.586
C08200=1089.350,-120.874,450.346,174.467,16.274,152.585
C08201=1089.356,-120.624,450.336,174.469,16.275,152.585
C08202=1089.362,-120.374,450.327,174.470,16.275,152.585
C08203=1089.369,-120.124,450.317,174.472,16.276,152.585
C08204=1089.375,-119.875,450.308,174.473,16.276,152.585
C08205=1089.381,-119.625,450.298,174.474,16.277,152.584
C08206=1089.386,-119.376,450.289,174.476,16.277,152.584
C08207=1089.392,-119.125,450.280,174.477,16.277,152.584
C08208=1089.399,-118.875,450.270,174.479,16.278,152.584
C08209=1089.405,-118.626,450.262,174.481,16.279,152.583
C08210=1089.412,-118.376,450.252,174.482,16.279,152.583
C08211=1089.418,-118.126,450.242,174.484,16.280,152.583
C08212=1089.424,-117.877,450.233,174.486,16.280,152.583
C08213=1089.430,-117.627,450.223,174.487,16.280,152.582
C08214=1089.436,-117.377,450.214,174.489,16.281,152.582
C08215=1089.442,-117.128,450.204,174.491,16.282,152.582
C08216=1089.448,-116.878,450.195,174.492,16.282,152.582
C08217=1089.454,-116.628,450.185,174.494,16.283,152.582
C08218=1089.460,-116.378,450.176,174.495,16.283,152.581
C08219=1089.466,-116.128,450.167,174.496,16.284,152.581
C08220=1089.472,-115.878,450.157,174.498,16.285,152.581
C08221=1089.479,-115.628,450.148,174.500,16.285,152.581
C08222=1089.485,-115.379,450.138,174.501,16.285,152.581
C08223=1089.491,-115.129,450.129,174.503,16.286,152.580
C08224=1089.497,-114.879,450.119,174.505,16.287,152.580
C08225=1089.503,-114.630,450.110,174.506,16.287,152.580
C08226=1089.509,-114.380,450.100,174.508,16.288,152.580
C08227=1089.515,-114.130,450.091,174.509,16.289,152.580
C08228=1089.521,-113.881,450.081,174.510,16.289,152.579
C08229=1089.527,-113.631,450.072,174.512,16.290,152.579
C08230=1089.534,-113.361,450.062,174.514,16.290,152.579
C08231=1089.541,-113.092,450.051,174.516,16.291,152.579
C08232=1089.547,-112.822,450.041,174.518,16.292,152.578
C08233=1089.554,-112.552,450.030,174.519,16.292,152.578
C08234=1089.560,-112.303,450.021,174.521,16.293,152.578
C08235=1089.566,-112.053,450.012,174.522,16.294,152.578
C08236=1089.572,-111.804,450.002,174.524,16.294,152.578
C08237=1089.579,-111.554,449.993,174.525,16.294,152.577
C08238=1089.584,-111.304,449.982,174.527,16.295,152.577
C08239=1089.590,-111.054,449.972,174.529,16.296,152.577
C08240=1089.597,-110.805,449.963,174.530,16.296,152.577
C08241=1089.603,-110.555,449.953,174.532,16.297,152.577
C08242=1089.609,-110.305,449.943,174.534,16.298,152.576
C08243=1089.615,-110.055,449.934,174.535,16.298,152.576
C08244=1089.621,-109.805,449.924,174.536,16.299,152.576
C08245=1089.627,-109.556,449.915,174.538,16.300,152.576
C08246=1089.634,-109.306,449.905,174.539,16.300,152.576
C08247=1089.640,-109.056,449.896,174.541,16.301,152.575
C08248=1089.646,-108.806,449.886,174.543,16.301,152.575
C08249=1089.652,-108.557,449.876,174.545,16.302,152.575
C08250=1089.658,-108.307,449.866,174.546,16.303,152.575
C08251=1089.664,-108.057,449.856,174.548,16.303,152.575
C08252=1089.670,-107.807,449.846,174.549,16.304,152.574
C08253=1089.676,-107.558,449.837,174.550,16.304,152.574
C08254=1089.683,-107.308,449.827,174.552,16.305,152.574
C08255=1089.689,-107.058,449.818,174.554,16.306,152.574
C08256=1089.695,-106.809,449.807,174.556,16.307,152.574
C08257=1089.701,-106.559,449.797,174.557,16.307,152.574
C08258=1089.707,-106.309,449.788,174.558,16.308,152.573
C08259=1089.713,-106.059,449.778,174.560,16.309,152.573
C08260=1089.719,-105.809,449.769,174.561,16.309,152.573
C08261=1089.725,-105.560,449.759,174.563,16.310,152.573
C08262=1089.731,-105.311,449.749,174.565,16.311,152.573
C08263=1089.737,-105.061,449.739,174.567,16.312,152.572
C08264=1089.743,-104.811,449.729,174.568,16.312,152.572
C08265=1089.749,-104.561,449.720,174.569,16.313,152.572
C08266=1089.755,-104.312,449.709,174.571,16.313,152.572
C08267=1089.761,-104.062,449.699,174.573,16.314,152.572
C08268=1089.767,-103.812,449.690,174.574,16.314,152.571
C08269=1089.773,-103.562,449.680,174.576,16.316,152.571
C08270=1089.779,-103.313,449.671,174.577,16.316,152.571
C08271=1089.785,-103.063,449.660,174.579,16.317,152.571
C08272=1089.791,-102.813,449.650,174.580,16.317,152.571
C08273=1089.798,-102.564,449.641,174.582,16.319,152.571
C08274=1089.803,-102.314,449.630,174.584,16.319,152.570
C08275=1089.810,-102.064,449.620,174.585,16.320,152.570
C08276=1089.816,-101.814,449.610,174.586,16.320,152.570
C08277=1089.822,-101.564,449.601,174.588,16.321,152.570
C08278=1089.828,-101.314,449.590,174.590,16.322,152.570
C08279=1089.834,-101.065,449.580,174.592,16.323,152.569
C08280=1089.840,-100.815,449.571,174.593,16.323,152.569
C08281=1089.847,-100.566,449.560,174.595,16.324,152.569
C08282=1089.852,-100.316,449.550,174.596,16.325,152.569
C08283=1089.859,-100.066,449.541,174.598,16.326,152.569
C08284=1089.865,-99.817,449.530,174.599,16.326,152.569
C08285=1089.870,-99.567,449.520,174.601,16.327,152.568
C08286=1089.877,-99.317,449.511,174.602,16.328,152.568
C08287=1089.883,-99.068,449.500,174.604,16.329,152.568
C08288=1089.889,-98.817,449.490,174.605,16.329,152.568
C08289=1089.895,-98.568,449.481,174.607,16.330,152.568
C08290=1089.901,-98.318,449.470,174.609,16.331,152.567
C08291=1089.907,-98.069,449.461,174.611,16.331,152.567
C08292=1089.913,-97.819,449.451,174.612,16.333,152.567
C08293=1089.919,-97.569,449.440,174.613,16.333,152.567
C08294=1089.926,-97.293,449.429,174.615,16.334,152.567
C08295=1089.932,-97.018,449.418,174.617,16.335,152.567
C08296=1089.939,-96.741,449.407,174.619,16.336,152.566
C08297=1089.945,-96.465,449.396,174.620,16.337,152.566
C08298=1089.952,-96.216,449.385,174.622,16.337,152.566
C08299=1089.957,-95.966,449.375,174.624,16.338,152.566
C08300=1089.964,-95.716,449.365,174.625,16.340,152.566
C08301=1089.970,-95.466,449.354,174.626,16.340,152.566
C08302=1089.976,-95.216,449.345,174.628,16.341,152.565
C08303=1089.982,-94.966,449.334,174.630,16.341,152.565
C08304=1089.988,-94.717,449.324,174.632,16.342,152.565
C08305=1089.994,-94.467,449.314,174.633,16.344,152.565
C08306=1090.000,-94.217,449.304,174.634,16.344,152.565
C08307=1090.005,-93.968,449.293,174.636,16.345,152.565
C08308=1090.012,-93.718,449.284,174.638,16.345,152.564
C08309=1090.017,-93.469,449.273,174.639,16.347,152.564
C08310=1090.024,-93.219,449.263,174.641,16.348,152.564
C08311=1090.029,-92.969,449.252,174.642,16.348,152.564
C08312=1090.035,-92.720,449.243,174.644,16.349,152.564
C08313=1090.041,-92.470,449.232,174.645,16.350,152.564
C08314=1090.048,-92.220,449.222,174.647,16.351,152.563
C08315=1090.054,-91.970,449.211,174.649,16.352,152.563
C08316=1090.060,-91.720,449.201,174.650,16.352,152.563
C08317=1090.066,-91.471,449.191,174.652,16.353,152.563
C08318=1090.072,-91.221,449.181,174.653,16.354,152.563
C08319=1090.078,-90.971,449.170,174.655,16.355,152.563
C08320=1090.083,-90.721,449.160,174.657,16.356,152.563
C08321=1090.089,-90.472,449.150,174.658,16.356,152.562
C08322=1090.095,-90.222,449.139,174.659,16.357,152.562
C08323=1090.102,-89.972,449.129,174.661,16.358,152.562
C08324=1090.108,-89.723,449.118,174.663,16.359,152.562
C08325=1090.114,-89.473,449.108,174.665,16.360,152.562
C08326=1090.120,-89.223,449.098,174.666,16.361,152.562
C08327=1090.126,-88.974,449.088,174.667,16.362,152.562
C08328=1090.132,-88.724,449.077,174.669,16.363,152.561
C08329=1090.138,-88.475,449.067,174.671,16.363,152.561
C08330=1090.144,-88.224,449.056,174.672,16.364,152.561
C08331=1090.150,-87.975,449.045,174.674,16.366,152.561
C08332=1090.156,-87.725,449.036,174.675,16.366,152.561
C08333=1090.162,-87.475,449.025,174.677,16.367,152.561
C08334=1090.168,-87.226,449.015,174.678,16.368,152.561
C08335=1090.174,-86.976,449.005,174.680,16.368,152.560
C08336=1090.180,-86.726,448.993,174.682,16.370,152.560
C08337=1090.186,-86.477,448.983,174.683,16.371,152.560
C08338=1090.192,-86.227,448.973,174.685,16.371,152.560
C08339=1090.198,-85.977,448.963,174.686,16.372,152.560
C08340=1090.204,-85.728,448.952,174.688,16.373,152.560
C08341=1090.211,-85.477,448.942,174.690,16.374,152.559
C08342=1090.217,-85.228,448.931,174.691,16.375,152.559
C08343=1090.222,-84.978,448.920,174.693,16.376,152.559
C08344=1090.228,-84.729,448.910,174.694,16.377,152.559
C08345=1090.234,-84.479,448.900,174.695,16.377,152.559
C08346=1090.241,-84.229,448.888,174.697,16.378,152.559
C08347=1090.247,-83.980,448.878,174.699,16.379,152.559
C08348=1090.252,-83.730,448.868,174.701,16.380,152.558
C08349=1090.259,-83.480,448.858,174.702,16.381,152.558
C08350=1090.265,-83.230,448.846,174.704,16.382,152.558
C08351=1090.271,-82.981,448.835,174.705,16.383,152.558
C08352=1090.277,-82.731,448.826,174.707,16.383,152.558
C08353=1090.283,-82.482,448.815,174.708,16.385,152.558
C08354=1090.289,-82.231,448.804,174.710,16.386,152.558
C08355=1090.296,-81.982,448.793,174.712,16.386,152.557
C08356=1090.301,-81.732,448.783,174.713,16.387,152.557
C08357=1090.308,-81.483,448.773,174.715,16.389,152.557
C08358=1090.314,-81.209,448.761,174.717,16.390,152.557
C08359=1090.321,-80.935,448.750,174.718,16.390,152.557
C08360=1090.328,-80.661,448.737,174.720,16.391,152.557
C08361=1090.335,-80.388,448.726,174.722,16.393,152.557
C08362=1090.340,-80.138,448.715,174.724,16.393,152.556
C08363=1090.347,-79.888,448.705,174.725,16.394,152.556
C08364=1090.352,-79.639,448.694,174.727,16.395,152.556
C08365=1090.359,-79.389,448.683,174.728,16.396,152.556
C08366=1090.364,-79.139,448.672,174.729,16.397,152.556
C08367=1090.370,-78.890,448.661,174.731,16.398,152.556
C08368=1090.376,-78.640,448.650,174.733,16.399,152.555
C08369=1090.383,-78.390,448.641,174.734,16.400,152.555
C08370=1090.388,-78.140,448.630,174.736,16.401,152.555
C08371=1090.394,-77.891,448.619,174.738,16.402,152.555
C08372=1090.400,-77.641,448.608,174.739,16.403,152.555
C08373=1090.406,-77.391,448.597,174.740,16.404,152.555
C08374=1090.413,-77.142,448.586,174.742,16.405,152.555
C08375=1090.418,-76.892,448.575,174.744,16.406,152.555
C08376=1090.424,-76.643,448.565,174.745,16.407,152.555
C08377=1090.431,-76.393,448.553,174.747,16.408,152.554
C08378=1090.436,-76.143,448.543,174.748,16.409,152.554
C08379=1090.442,-75.893,448.532,174.750,16.410,152.554
C08380=1090.447,-75.644,448.521,174.752,16.411,152.554
C08381=1090.455,-75.394,448.511,174.754,16.412,152.554
C08382=1090.460,-75.144,448.500,174.755,16.413,152.554
C08383=1090.466,-74.895,448.489,174.756,16.414,152.554
C08384=1090.472,-74.645,448.478,174.758,16.415,152.554
C08385=1090.478,-74.395,448.467,174.759,16.416,152.553
C08386=1090.484,-74.146,448.456,174.761,16.417,152.553
C08387=1090.490,-73.895,448.445,174.763,16.418,152.553
C08388=1090.496,-73.646,448.434,174.764,16.419,152.553
C08389=1090.502,-73.396,448.423,174.766,16.420,152.553
C08390=1090.507,-73.147,448.412,174.768,16.421,152.553
C08391=1090.513,-72.898,448.401,174.769,16.422,152.553
C08392=1090.519,-72.647,448.390,174.771,16.423,152.553
C08393=1090.525,-72.398,448.379,174.773,16.424,152.552
C08394=1090.531,-72.148,448.368,174.774,16.426,152.552
C08395=1090.537,-71.898,448.357,174.775,16.426,152.552
C08396=1090.543,-71.649,448.346,174.777,16.427,152.552
C08397=1090.549,-71.399,448.335,174.778,16.428,152.552
C08398=1090.554,-71.150,448.324,174.780,16.429,152.552
C08399=1090.561,-70.899,448.313,174.781,16.431,152.552
C08400=1090.567,-70.650,448.302,174.783,16.432,152.552
C08401=1090.572,-70.401,448.291,174.785,16.433,152.552
C08402=1090.578,-70.151,448.281,174.786,16.434,152.552
C08403=1090.584,-69.901,448.269,174.788,16.435,152.551
C08404=1090.589,-69.651,448.258,174.790,16.436,152.551
C08405=1090.595,-69.402,448.247,174.791,16.437,152.551
C08406=1090.601,-69.151,448.236,174.793,16.438,152.551
C08407=1090.607,-68.902,448.225,174.795,16.439,152.551
C08408=1090.613,-68.653,448.213,174.796,16.440,152.551
C08409=1090.620,-68.403,448.202,174.798,16.441,152.551
C08410=1090.625,-68.153,448.191,174.800,16.443,152.550
C08411=1090.631,-67.904,448.180,174.800,16.443,152.550
C08412=1090.637,-67.654,448.169,174.802,16.444,152.550
C08413=1090.643,-67.404,448.158,174.804,16.445,152.550
C08414=1090.648,-67.154,448.147,174.805,16.446,152.550
C08415=1090.654,-66.904,448.135,174.807,16.448,152.550
C08416=1090.661,-66.655,448.124,174.808,16.449,152.550
C08417=1090.666,-66.406,448.113,174.810,16.450,152.550
C08418=1090.673,-66.156,448.102,174.812,16.451,152.550
C08419=1090.678,-65.906,448.091,174.813,16.452,152.550
C08420=1090.684,-65.657,448.080,174.815,16.453,152.549
C08421=1090.690,-65.406,448.069,174.817,16.454,152.549
C08422=1090.696,-65.135,448.056,174.818,16.455,152.549
C08423=1090.703,-64.864,448.044,174.820,16.457,152.549
C08424=1090.710,-64.592,448.032,174.821,16.458,152.549
C08425=1090.716,-64.321,448.020,174.823,16.459,152.549
C08426=1090.722,-64.071,448.008,174.825,16.460,152.549
C08427=1090.727,-63.821,447.997,174.826,16.461,152.549
C08428=1090.733,-63.572,447.985,174.828,16.462,152.549
C08429=1090.740,-63.322,447.974,174.829,16.463,152.549
C08430=1090.746,-63.072,447.963,174.831,16.465,152.548
C08431=1090.752,-62.822,447.952,174.833,16.466,152.548
C08432=1090.758,-62.573,447.940,174.834,16.467,152.548
C08433=1090.763,-62.324,447.929,174.836,16.468,152.548
C08434=1090.769,-62.073,447.918,174.838,16.469,152.548
C08435=1090.775,-61.824,447.907,174.839,16.470,152.548
C08436=1090.782,-61.574,447.895,174.841,16.471,152.548
C08437=1090.787,-61.325,447.884,174.842,16.472,152.548
C08438=1090.794,-61.075,447.873,174.844,16.474,152.548
C08439=1090.799,-60.825,447.860,174.846,16.475,152.547
C08440=1090.805,-60.575,447.849,174.847,16.476,152.547
C08441=1090.811,-60.326,447.838,174.849,16.477,152.547
C08442=1090.817,-60.076,447.827,174.850,16.478,152.547
C08443=1090.824,-59.827,447.815,174.852,16.479,152.547
C08444=1090.829,-59.577,447.804,174.854,16.480,152.547
C08445=1090.835,-59.327,447.792,174.855,16.481,152.547
C08446=1090.841,-59.078,447.781,174.857,16.483,152.547
C08447=1090.847,-58.828,447.770,174.859,16.484,152.547
C08448=1090.853,-58.579,447.758,174.860,16.485,152.546
C08449=1090.859,-58.328,447.746,174.862,16.486,152.546
C08450=1090.865,-58.079,447.736,174.863,16.487,152.546
C08451=1090.871,-57.829,447.724,174.865,16.488,152.546
C08452=1090.877,-57.580,447.713,174.867,16.489,152.546
C08453=1090.883,-57.330,447.700,174.868,16.490,152.546
C08454=1090.889,-57.080,447.689,174.870,16.492,152.546
C08455=1090.895,-56.830,447.678,174.872,16.493,152.546
C08456=1090.901,-56.581,447.666,174.873,16.494,152.546
C08457=1090.907,-56.331,447.655,174.875,16.495,152.546
C08458=1090.913,-56.082,447.643,174.876,16.496,152.545
C08459=1090.919,-55.832,447.632,174.878,16.497,152.545
C08460=1090.925,-55.583,447.620,174.880,16.498,152.545
C08461=1090.931,-55.333,447.609,174.881,16.499,152.545
C08462=1090.937,-55.083,447.597,174.883,16.501,152.545
C08463=1090.943,-54.833,447.586,174.884,16.502,152.545
C08464=1090.949,-54.583,447.574,174.886,16.503,152.545
C08465=1090.955,-54.334,447.563,174.888,16.504,152.545
C08466=1090.961,-54.084,447.551,174.889,16.505,152.545
C08467=1090.967,-53.835,447.539,174.891,16.506,152.544
C08468=1090.973,-53.585,447.528,174.893,16.507,152.544
C08469=1090.979,-53.335,447.516,174.894,16.509,152.544
C08470=1090.985,-53.085,447.505,174.896,16.510,152.544
C08471=1090.991,-52.836,447.493,174.897,16.511,152.544
C08472=1090.998,-52.587,447.481,174.899,16.512,152.544
C08473=1091.003,-52.336,447.469,174.901,16.513,152.544
C08474=1091.009,-52.087,447.458,174.902,16.514,152.544
C08475=1091.016,-51.837,447.446,174.904,16.515,152.544
C08476=1091.021,-51.588,447.434,174.905,16.516,152.544
C08477=1091.027,-51.338,447.423,174.907,16.518,152.543
C08478=1091.034,-51.088,447.411,174.909,16.519,152.543
C08479=1091.040,-50.839,447.399,174.910,16.520,152.543
C08480=1091.046,-50.589,447.388,174.912,16.521,152.543
C08481=1091.052,-50.340,447.376,174.913,16.523,152.543
C08482=1091.057,-50.090,447.364,174.915,16.524,152.543
C08483=1091.063,-49.841,447.352,174.917,16.525,152.543
C08484=1091.069,-49.590,447.341,174.918,16.526,152.543
C08485=1091.076,-49.341,447.329,174.920,16.527,152.543
C08486=1091.081,-49.071,447.315,174.922,16.529,152.543
C08487=1091.088,-48.800,447.303,174.924,16.530,152.542
C08488=1091.094,-48.530,447.290,174.925,16.532,152.543
C08489=1091.101,-48.260,447.278,174.927,16.533,152.542
C08490=1091.106,-48.011,447.266,174.928,16.534,152.542
C08491=1091.113,-47.761,447.254,174.930,16.535,152.542
C08492=1091.118,-47.511,447.242,174.932,16.536,152.542
C08493=1091.124,-47.261,447.230,174.933,16.537,152.542
C08494=1091.130,-47.012,447.218,174.935,16.538,152.542
C08495=1091.135,-46.762,447.206,174.937,16.541,152.542
C08496=1091.142,-46.512,447.194,174.939,16.542,152.542
C08497=1091.147,-46.263,447.182,174.940,16.543,152.542
C08498=1091.154,-46.013,447.171,174.942,16.544,152.542
C08499=1091.160,-45.763,447.158,174.943,16.545,152.542
C08500=1091.166,-45.514,447.147,174.945,16.546,152.541
C08501=1091.171,-45.264,447.134,174.947,16.547,152.541
C08502=1091.176,-45.015,447.123,174.948,16.549,152.541
C08503=1091.183,-44.765,447.111,174.950,16.550,152.541
C08504=1091.189,-44.515,447.098,174.951,16.551,152.541
C08505=1091.195,-44.266,447.087,174.953,16.552,152.541
C08506=1091.201,-44.016,447.075,174.955,16.553,152.541
C08507=1091.206,-43.767,447.062,174.956,16.555,152.541
C08508=1091.213,-43.517,447.050,174.958,16.556,152.541
C08509=1091.219,-43.267,447.038,174.959,16.557,152.541
C08510=1091.224,-43.018,447.027,174.961,16.558,152.541
C08511=1091.230,-42.768,447.014,174.963,16.560,152.541
C08512=1091.236,-42.518,447.002,174.965,16.561,152.540
C08513=1091.242,-42.269,446.990,174.966,16.562,152.540
C08514=1091.248,-42.019,446.978,174.968,16.564,152.540
C08515=1091.254,-41.769,446.966,174.970,16.565,152.540
C08516=1091.260,-41.520,446.954,174.971,16.566,152.540
C08517=1091.266,-41.270,446.942,174.973,16.567,152.540
C08518=1091.272,-41.020,446.930,174.974,16.569,152.540
C08519=1091.278,-40.771,446.918,174.976,16.570,152.540
C08520=1091.283,-40.521,446.905,174.977,16.571,152.540
C08521=1091.290,-40.271,446.894,174.979,16.572,152.540
C08522=1091.295,-40.022,446.882,174.981,16.573,152.540
C08523=1091.301,-39.772,446.869,174.982,16.574,152.539
C08524=1091.308,-39.522,446.857,174.984,16.576,152.539
C08525=1091.313,-39.273,446.845,174.986,16.577,152.539
C08526=1091.319,-39.023,446.832,174.988,16.579,152.539
C08527=1091.326,-38.774,446.820,174.989,16.580,152.539
C08528=1091.331,-38.525,446.808,174.991,16.581,152.539
C08529=1091.337,-38.275,446.796,174.992,16.582,152.539
C08530=1091.342,-38.024,446.784,174.994,16.584,152.539
C08531=1091.348,-37.775,446.772,174.995,16.585,152.539
C08532=1091.354,-37.525,446.760,174.997,16.586,152.539
C08533=1091.360,-37.276,446.747,174.999,16.587,152.539
C08534=1091.366,-37.026,446.735,175.000,16.589,152.539
C08535=1091.371,-36.777,446.722,175.002,16.590,152.539
C08536=1091.378,-36.527,446.710,175.004,16.591,152.538
C08537=1091.383,-36.278,446.698,175.006,16.593,152.538
C08538=1091.389,-36.028,446.686,175.007,16.594,152.538
C08539=1091.395,-35.778,446.673,175.009,16.595,152.538
C08540=1091.401,-35.528,446.661,175.010,16.596,152.538
C08541=1091.406,-35.279,446.648,175.012,16.598,152.538
C08542=1091.413,-35.029,446.636,175.013,16.599,152.538
C08543=1091.419,-34.779,446.624,175.015,16.600,152.538
C08544=1091.424,-34.530,446.612,175.016,16.602,152.538
C08545=1091.430,-34.280,446.599,175.019,16.603,152.538
C08546=1091.436,-34.031,446.587,175.020,16.604,152.538
C08547=1091.442,-33.781,446.574,175.022,16.605,152.538
C08548=1091.447,-33.531,446.562,175.024,16.607,152.537
C08549=1091.454,-33.282,446.550,175.025,16.608,152.538
C08550=1091.460,-33.012,446.536,175.027,16.609,152.537
C08551=1091.467,-32.742,446.523,175.029,16.611,152.537
C08552=1091.472,-32.473,446.509,175.031,16.612,152.537
C08553=1091.479,-32.203,446.496,175.032,16.613,152.537
C08554=1091.485,-31.953,446.484,175.034,16.615,152.537
C08555=1091.491,-31.703,446.471,175.035,16.616,152.537
C08556=1091.497,-31.454,446.458,175.038,16.618,152.537
C08557=1091.503,-31.204,446.446,175.039,16.619,152.537
C08558=1091.508,-30.955,446.433,175.041,16.620,152.537
C08559=1091.514,-30.705,446.421,175.042,16.622,152.537
C08560=1091.520,-30.455,446.408,175.044,16.623,152.537
C08561=1091.526,-30.206,446.396,175.046,16.624,152.537
C08562=1091.532,-29.956,446.383,175.047,16.625,152.536
C08563=1091.538,-29.706,446.371,175.049,16.626,152.536
C08564=1091.544,-29.457,446.358,175.051,16.628,152.536
C08565=1091.550,-29.207,446.345,175.052,16.629,152.536
C08566=1091.556,-28.958,446.333,175.054,16.631,152.536
C08567=1091.562,-28.708,446.321,175.056,16.632,152.536
C08568=1091.567,-28.458,446.308,175.057,16.633,152.536
C08569=1091.574,-28.209,446.295,175.059,16.634,152.536
C08570=1091.580,-27.959,446.282,175.060,16.636,152.536
C08571=1091.585,-27.709,446.270,175.062,16.637,152.536
C08572=1091.591,-27.460,446.258,175.064,16.638,152.536
C08573=1091.597,-27.210,446.245,175.066,16.640,152.536
C08574=1091.603,-26.961,446.232,175.068,16.641,152.535
C08575=1091.609,-26.711,446.219,175.069,16.642,152.535
C08576=1091.615,-26.461,446.207,175.071,16.643,152.535
C08577=1091.620,-26.212,446.195,175.072,16.645,152.535
C08578=1091.626,-25.962,446.181,175.074,16.646,152.535
C08579=1091.632,-25.713,446.169,175.076,16.648,152.535
C08580=1091.638,-25.463,446.156,175.078,16.649,152.535
C08581=1091.644,-25.213,446.144,175.079,16.650,152.535
C08582=1091.650,-24.964,446.131,175.081,16.651,152.535
C08583=1091.655,-24.714,446.118,175.082,16.653,152.535
C08584=1091.661,-24.464,446.105,175.084,16.654,152.535
C08585=1091.667,-24.215,446.092,175.085,16.655,152.535
C08586=1091.673,-23.965,446.079,175.088,16.657,152.535
C08587=1091.679,-23.715,446.067,175.089,16.658,152.535
C08588=1091.684,-23.467,446.054,175.091,16.660,152.535
C08589=1091.690,-23.217,446.041,175.092,16.661,152.534
C08590=1091.696,-22.967,446.029,175.094,16.662,152.534
C08591=1091.702,-22.717,446.015,175.095,16.664,152.534
C08592=1091.707,-22.467,446.002,175.098,16.665,152.534
C08593=1091.713,-22.217,445.990,175.099,16.666,152.534
C08594=1091.720,-21.968,445.976,175.101,16.667,152.534
C08595=1091.725,-21.719,445.964,175.102,16.669,152.534
C08596=1091.731,-21.469,445.952,175.104,16.670,152.534
C08597=1091.737,-21.220,445.938,175.106,16.671,152.534
C08598=1091.742,-20.970,445.925,175.108,16.673,152.534
C08599=1091.748,-20.720,445.912,175.109,16.675,152.534
C08600=1091.754,-20.471,445.899,175.111,16.676,152.534
C08601=1091.760,-20.221,445.887,175.113,16.677,152.534
C08602=1091.766,-19.971,445.874,175.114,16.678,152.533
C08603=1091.772,-19.722,445.861,175.116,16.679,152.533
C08604=1091.777,-19.473,445.847,175.118,16.681,152.533
C08605=1091.783,-19.223,445.835,175.120,16.682,152.533
C08606=1091.789,-18.974,445.822,175.121,16.684,152.533
C08607=1091.795,-18.724,445.809,175.123,16.685,152.533
C08608=1091.801,-18.474,445.796,175.124,16.686,152.533
C08609=1091.807,-18.224,445.783,175.126,16.688,152.533
C08610=1091.813,-17.975,445.769,175.128,16.689,152.533
C08611=1091.819,-17.725,445.757,175.130,16.690,152.533
C08612=1091.825,-17.476,445.744,175.131,16.691,152.533
C08613=1091.831,-17.226,445.731,175.133,16.693,152.533
C08614=1091.836,-16.955,445.717,175.135,16.695,152.533
C08615=1091.843,-16.685,445.702,175.137,16.696,152.532
C08616=1091.850,-16.414,445.688,175.138,16.697,152.532
C08617=1091.856,-16.144,445.674,175.141,16.699,152.532
C08618=1091.862,-15.894,445.661,175.142,16.700,152.532
C08619=1091.867,-15.644,445.648,175.144,16.701,152.532
C08620=1091.873,-15.395,445.635,175.145,16.703,152.532
C08621=1091.879,-15.145,445.622,175.147,16.704,152.532
C08622=1091.885,-14.896,445.609,175.149,16.706,152.532
C08623=1091.891,-14.645,445.596,175.151,16.707,152.532
C08624=1091.897,-14.396,445.583,175.152,16.708,152.532
C08625=1091.902,-14.147,445.569,175.154,16.709,152.532
C08626=1091.908,-13.897,445.556,175.155,16.711,152.532
C08627=1091.914,-13.647,445.543,175.158,16.713,152.532
C08628=1091.920,-13.397,445.530,175.159,16.714,152.532
C08629=1091.926,-13.148,445.516,175.161,16.715,152.531
C08630=1091.932,-12.899,445.503,175.162,16.717,152.531
C08631=1091.937,-12.649,445.490,175.164,16.718,152.531
C08632=1091.943,-12.399,445.477,175.166,16.719,152.531
C08633=1091.949,-12.150,445.463,175.168,16.720,152.531
C08634=1091.955,-11.900,445.450,175.169,16.722,152.531
C08635=1091.960,-11.650,445.436,175.171,16.723,152.531
C08636=1091.967,-11.401,445.423,175.173,16.724,152.531
C08637=1091.972,-11.151,445.411,175.175,16.726,152.531
C08638=1091.978,-10.902,445.397,175.176,16.728,152.531
C08639=1091.984,-10.652,445.383,175.178,16.729,152.531
C08640=1091.989,-10.402,445.370,175.180,16.730,152.531
C08641=1091.996,-10.153,445.357,175.181,16.731,152.531
C08642=1092.001,-9.903,445.343,175.183,16.733,152.531
C08643=1092.007,-9.654,445.330,175.185,16.734,152.530
C08644=1092.013,-9.404,445.317,175.187,16.735,152.530
C08645=1092.019,-9.155,445.304,175.188,16.737,152.530
C08646=1092.025,-8.905,445.290,175.190,16.738,152.530
C08647=1092.030,-8.656,445.276,175.192,16.740,152.530
C08648=1092.036,-8.406,445.264,175.194,16.741,152.530
C08649=1092.042,-8.156,445.250,175.195,16.742,152.530
C08650=1092.048,-7.907,445.237,175.197,16.743,152.530
C08651=1092.053,-7.657,445.223,175.199,16.746,152.530
C08652=1092.060,-7.408,445.210,175.201,16.747,152.530
C08653=1092.065,-7.158,445.196,175.202,16.748,152.530
C08654=1092.071,-6.909,445.183,175.204,16.749,152.530
C08655=1092.076,-6.659,445.169,175.205,16.750,152.530
C08656=1092.083,-6.410,445.156,175.208,16.752,152.530
C08657=1092.088,-6.160,445.142,175.209,16.753,152.529
C08658=1092.094,-5.910,445.130,175.211,16.754,152.529
C08659=1092.099,-5.661,445.116,175.212,16.756,152.529
C08660=1092.106,-5.411,445.102,175.215,16.757,152.529
C08661=1092.112,-5.161,445.088,175.216,16.759,152.529
C08662=1092.118,-4.912,445.075,175.218,16.760,152.529
C08663=1092.123,-4.662,445.061,175.219,16.761,152.529
C08664=1092.130,-4.413,445.048,175.221,16.762,152.529
C08665=1092.135,-4.164,445.034,175.224,16.764,152.529
C08666=1092.141,-3.914,445.021,175.225,16.765,152.529
C08667=1092.147,-3.664,445.008,175.226,16.767,152.529
C08668=1092.153,-3.415,444.994,175.228,16.768,152.529
C08669=1092.159,-3.165,444.980,175.231,16.770,152.528
C08670=1092.164,-2.915,444.966,175.232,16.771,152.528
C08671=1092.171,-2.666,444.953,175.233,16.772,152.528
C08672=1092.176,-2.416,444.939,175.235,16.773,152.528
C08673=1092.181,-2.167,444.925,175.238,16.775,152.528
C08674=1092.188,-1.917,444.912,175.239,16.776,152.528
C08675=1092.193,-1.668,444.898,175.240,16.778,152.528
C08676=1092.199,-1.418,444.884,175.242,16.779,152.528
C08677=1092.204,-1.169,444.870,175.245,16.781,152.528
C08678=1092.211,-0.897,444.855,175.246,16.782,152.528
C08679=1092.217,-0.624,444.841,175.248,16.783,152.528
C08680=1092.223,-0.352,444.826,175.250,16.785,152.528
C08681=1092.229,-0.080,444.811,175.252,16.786,152.528
C08682=1092.235,0.170,444.797,175.254,16.788,152.527
C08683=1092.241,0.419,444.783,175.255,16.790,152.527
C08684=1092.247,0.670,444.769,175.257,16.791,152.527
C08685=1092.252,0.919,444.755,175.259,16.792,152.527
C08686=1092.258,1.169,444.741,175.261,16.794,152.527
C08687=1092.264,1.418,444.728,175.262,16.795,152.527
C08688=1092.269,1.668,444.714,175.264,16.796,152.527
C08689=1092.275,1.917,444.700,175.266,16.797,152.527
C08690=1092.280,2.167,444.687,175.268,16.799,152.527
C08691=1092.287,2.416,444.673,175.269,16.801,152.527
C08692=1092.293,2.666,444.659,175.271,16.802,152.527
C08693=1092.298,2.915,444.645,175.273,16.803,152.527
C08694=1092.304,3.165,444.631,175.275,16.805,152.527
C08695=1092.309,3.414,444.617,175.277,16.806,152.526
C08696=1092.316,3.664,444.604,175.278,16.807,152.527
C08697=1092.321,3.913,444.590,175.280,16.809,152.526
C08698=1092.327,4.164,444.575,175.282,16.810,152.526
C08699=1092.333,4.413,444.562,175.284,16.811,152.526
C08700=1092.338,4.663,444.548,175.285,16.813,152.526
C08701=1092.345,4.911,444.534,175.287,16.815,152.526
C08702=1092.350,5.161,444.520,175.289,16.816,152.526
C08703=1092.356,5.410,444.506,175.291,16.817,152.526
C08704=1092.362,5.661,444.492,175.292,16.818,152.526
C08705=1092.367,5.910,444.478,175.295,16.820,152.526
C08706=1092.373,6.159,444.463,175.296,16.821,152.526
C08707=1092.379,6.409,444.450,175.298,16.823,152.526
C08708=1092.385,6.659,444.436,175.299,16.824,152.526
C08709=1092.391,6.908,444.422,175.302,16.825,152.525
C08710=1092.396,7.158,444.408,175.303,16.826,152.525
C08711=1092.402,7.407,444.394,175.305,16.828,152.525
C08712=1092.407,7.656,444.380,175.307,16.829,152.525
C08713=1092.414,7.907,444.365,175.309,16.831,152.525
C08714=1092.420,8.156,444.352,175.310,16.832,152.525
C08715=1092.426,8.405,444.338,175.312,16.833,152.525
C08716=1092.431,8.655,444.324,175.314,16.835,152.525
C08717=1092.437,8.905,444.309,175.316,16.836,152.525
C08718=1092.443,9.154,444.295,175.318,16.837,152.525
C08719=1092.448,9.403,444.281,175.319,16.838,152.524
C08720=1092.454,9.654,444.267,175.321,16.840,152.524
C08721=1092.460,9.903,444.252,175.323,16.842,152.524
C08722=1092.466,10.152,444.239,175.325,16.843,152.524
C08723=1092.472,10.401,444.225,175.327,16.844,152.524
C08724=1092.478,10.651,444.210,175.329,16.846,152.524
C08725=1092.484,10.901,444.196,175.330,16.847,152.524
C08726=1092.489,11.150,444.182,175.332,16.848,152.524
C08727=1092.496,11.400,444.167,175.334,16.849,152.524
C08728=1092.501,11.649,444.154,175.336,16.851,152.524
C08729=1092.507,11.899,444.140,175.337,16.852,152.524
C08730=1092.512,12.148,444.125,175.340,16.854,152.524
C08731=1092.518,12.398,444.111,175.341,16.855,152.523
C08732=1092.524,12.647,444.096,175.343,16.856,152.523
C08733=1092.530,12.896,444.083,175.345,16.857,152.523
C08734=1092.536,13.147,444.069,175.347,16.859,152.523
C08735=1092.542,13.396,444.054,175.349,16.860,152.523
C08736=1092.548,13.646,444.040,175.350,16.861,152.523
C08737=1092.554,13.895,444.025,175.353,16.863,152.523
C08738=1092.560,14.145,444.012,175.354,16.864,152.523
C08739=1092.566,14.394,443.997,175.356,16.865,152.523
C08740=1092.571,14.644,443.983,175.357,16.867,152.523
C08741=1092.577,14.893,443.968,175.360,16.869,152.522
C08742=1092.583,15.167,443.952,175.361,16.870,152.522
C08743=1092.590,15.442,443.936,175.364,16.871,152.522
C08744=1092.596,15.716,443.921,175.365,16.872,152.522
C08745=1092.602,15.990,443.905,175.368,16.874,152.522
C08746=1092.608,16.240,443.890,175.369,16.875,152.522
C08747=1092.614,16.490,443.876,175.372,16.877,152.522
C08748=1092.619,16.738,443.862,175.373,16.879,152.522
C08749=1092.625,16.989,443.847,175.375,16.880,152.522
C08750=1092.631,17.238,443.833,175.376,16.881,152.522
C08751=1092.637,17.487,443.819,175.379,16.883,152.521
C08752=1092.642,17.737,443.803,175.381,16.884,152.521
C08753=1092.648,17.987,443.790,175.382,16.885,152.521
C08754=1092.654,18.236,443.775,175.385,16.886,152.521
C08755=1092.660,18.485,443.760,175.386,16.888,152.521
C08756=1092.665,18.735,443.746,175.388,16.889,152.521
C08757=1092.672,18.985,443.731,175.390,16.890,152.521
C08758=1092.677,19.234,443.717,175.392,16.892,152.521
C08759=1092.682,19.484,443.702,175.393,16.893,152.521
C08760=1092.689,19.733,443.687,175.396,16.895,152.521
C08761=1092.694,19.983,443.673,175.397,16.896,152.521
C08762=1092.701,20.232,443.658,175.399,16.897,152.520
C08763=1092.706,20.481,443.644,175.401,16.899,152.520
C08764=1092.712,20.731,443.630,175.403,16.900,152.520
C08765=1092.718,20.981,443.615,175.405,16.901,152.520
C08766=1092.723,21.230,443.601,175.407,16.903,152.520
C08767=1092.729,21.479,443.586,175.409,16.904,152.520
C08768=1092.734,21.729,443.571,175.410,16.905,152.520
C08769=1092.740,21.978,443.556,175.412,16.906,152.520
C08770=1092.746,22.229,443.542,175.414,16.908,152.520
C08771=1092.752,22.478,443.527,175.416,16.909,152.520
C08772=1092.757,22.727,443.512,175.417,16.911,152.520
C08773=1092.763,22.977,443.498,175.420,16.912,152.519
C08774=1092.769,23.226,443.483,175.421,16.913,152.519
C08775=1092.775,23.476,443.468,175.423,16.915,152.519
C08776=1092.780,23.725,443.453,175.425,16.916,152.519
C08777=1092.786,23.975,443.439,175.427,16.917,152.519
C08778=1092.792,24.224,443.424,175.429,16.918,152.519
C08779=1092.797,24.473,443.409,175.431,16.920,152.519
C08780=1092.804,24.723,443.394,175.433,16.921,152.519
C08781=1092.809,24.973,443.380,175.434,16.922,152.519
C08782=1092.816,25.222,443.365,175.437,16.924,152.518
C08783=1092.821,25.472,443.350,175.438,16.925,152.518
C08784=1092.827,25.721,443.335,175.441,16.927,152.518
C08785=1092.833,25.970,443.321,175.442,16.928,152.518
C08786=1092.838,26.220,443.305,175.444,16.929,152.518
C08787=1092.844,26.470,443.291,175.446,16.931,152.518
C08788=1092.850,26.719,443.276,175.448,16.932,152.518
C08789=1092.855,26.969,443.261,175.450,16.933,152.518
C08790=1092.862,27.218,443.246,175.452,16.935,152.518
C08791=1092.867,27.467,443.232,175.454,16.936,152.517
C08792=1092.873,27.717,443.216,175.455,16.937,152.517
C08793=1092.879,27.966,443.201,175.458,16.939,152.517
C08794=1092.884,28.217,443.187,175.459,16.940,152.517
C08795=1092.890,28.466,443.172,175.461,16.941,152.517
C08796=1092.896,28.715,443.157,175.463,16.943,152.517
C08797=1092.901,28.965,443.142,175.465,16.944,152.517
C08798=1092.908,29.214,443.127,175.467,16.945,152.517
C08799=1092.913,29.464,443.112,175.469,16.947,152.517
C08800=1092.919,29.713,443.097,175.471,16.948,152.516
C08801=1092.924,29.963,443.082,175.472,16.949,152.516
C08802=1092.930,30.212,443.067,175.475,16.951,152.516
C08803=1092.936,30.462,443.052,175.476,16.952,152.516
C08804=1092.941,30.710,443.037,175.479,16.953,152.516
C08805=1092.947,30.960,443.021,175.481,16.955,152.516
C08806=1092.954,31.236,443.005,175.482,16.956,152.516
C08807=1092.960,31.512,442.989,175.485,16.957,152.516
C08808=1092.966,31.788,442.972,175.487,16.959,152.515
C08809=1092.973,32.064,442.955,175.489,16.960,152.515
C08810=1092.978,32.313,442.940,175.491,16.962,152.515
C08811=1092.984,32.563,442.925,175.493,16.963,152.515
C08812=1092.989,32.812,442.910,175.494,16.964,152.515
C08813=1092.996,33.062,442.895,175.497,16.966,152.515
C08814=1093.001,33.311,442.880,175.498,16.967,152.515
C08815=1093.007,33.561,442.865,175.501,16.969,152.515
C08816=1093.012,33.810,442.849,175.502,16.970,152.515
C08817=1093.018,34.060,442.835,175.504,16.971,152.515
C08818=1093.024,34.308,442.819,175.507,16.972,152.514
C08819=1093.030,34.558,442.804,175.508,16.973,152.514
C08820=1093.036,34.808,442.788,175.510,16.974,152.514
C08821=1093.042,35.057,442.774,175.512,16.976,152.514
C08822=1093.047,35.307,442.758,175.514,16.977,152.514
C08823=1093.052,35.556,442.743,175.516,16.978,152.514
C08824=1093.059,35.806,442.728,175.518,16.980,152.514
C08825=1093.064,36.056,442.712,175.520,16.981,152.513
C08826=1093.070,36.304,442.697,175.522,16.983,152.513
C08827=1093.076,36.554,442.682,175.524,16.984,152.513
C08828=1093.082,36.803,442.667,175.526,16.985,152.513
C08829=1093.087,37.053,442.651,175.528,16.986,152.513
C08830=1093.093,37.303,442.636,175.530,16.987,152.513
C08831=1093.099,37.552,442.621,175.532,16.989,152.513
C08832=1093.105,37.801,442.605,175.534,16.990,152.513
C08833=1093.110,38.051,442.589,175.535,16.991,152.512
C08834=1093.116,38.300,442.575,175.538,16.993,152.512
C08835=1093.122,38.550,442.559,175.539,16.994,152.512
C08836=1093.127,38.799,442.544,175.541,16.995,152.512
C08837=1093.134,39.048,442.529,175.544,16.997,152.512
C08838=1093.139,39.298,442.513,175.545,16.998,152.512
C08839=1093.144,39.548,442.498,175.548,16.999,152.512
C08840=1093.150,39.798,442.482,175.549,17.000,152.512
C08841=1093.156,40.046,442.467,175.551,17.002,152.511
C08842=1093.162,40.296,442.451,175.554,17.003,152.511
C08843=1093.167,40.546,442.436,175.555,17.004,152.511
C08844=1093.173,40.794,442.420,175.558,17.006,152.511
C08845=1093.179,41.044,442.405,175.559,17.007,152.511
C08846=1093.185,41.294,442.390,175.561,17.008,152.511
C08847=1093.190,41.543,442.374,175.564,17.010,152.511
C08848=1093.196,41.793,442.358,175.565,17.011,152.510
C08849=1093.201,42.042,442.343,175.568,17.012,152.510
C08850=1093.207,42.291,442.327,175.569,17.014,152.510
C08851=1093.213,42.541,442.312,175.571,17.015,152.510
C08852=1093.218,42.790,442.297,175.574,17.016,152.510
C08853=1093.224,43.040,442.280,175.575,17.017,152.510
C08854=1093.230,43.289,442.265,175.578,17.019,152.510
C08855=1093.236,43.539,442.250,175.579,17.020,152.510
C08856=1093.241,43.788,442.234,175.581,17.021,152.509
C08857=1093.247,44.038,442.218,175.583,17.023,152.509
C08858=1093.252,44.286,442.202,175.585,17.023,152.509
C08859=1093.258,44.536,442.187,175.588,17.025,152.509
C08860=1093.264,44.786,442.171,175.589,17.026,152.509
C08861=1093.269,45.035,442.156,175.591,17.027,152.509
C08862=1093.275,45.285,442.140,175.593,17.029,152.509
C08863=1093.281,45.534,442.124,175.595,17.030,152.509
C08864=1093.286,45.784,442.109,175.597,17.032,152.508
C08865=1093.292,46.033,442.092,175.599,17.032,152.508
C08866=1093.297,46.283,442.077,175.602,17.034,152.508
C08867=1093.303,46.532,442.061,175.603,17.035,152.508
C08868=1093.308,46.782,442.045,175.605,17.036,152.508
C08869=1093.314,47.032,442.030,175.607,17.038,152.508
C08870=1093.321,47.306,442.013,175.610,17.040,152.508
C08871=1093.327,47.583,441.995,175.612,17.040,152.507
C08872=1093.333,47.858,441.977,175.614,17.042,152.507
C08873=1093.339,48.134,441.960,175.617,17.044,152.507
C08874=1093.345,48.383,441.944,175.618,17.045,152.507
C08875=1093.351,48.633,441.928,175.620,17.046,152.507
C08876=1093.356,48.882,441.912,175.623,17.047,152.507
C08877=1093.362,49.132,441.897,175.624,17.048,152.506
C08878=1093.367,49.381,441.881,175.627,17.050,152.506
C08879=1093.373,49.631,441.865,175.628,17.051,152.506
C08880=1093.378,49.880,441.849,175.631,17.052,152.506
C08881=1093.384,50.129,441.833,175.633,17.053,152.506
C08882=1093.390,50.379,441.817,175.634,17.055,152.506
C08883=1093.396,50.628,441.801,175.637,17.056,152.506
C08884=1093.401,50.877,441.786,175.639,17.057,152.505
C08885=1093.407,51.127,441.770,175.641,17.059,152.505
C08886=1093.413,51.376,441.753,175.643,17.060,152.505
C08887=1093.419,51.626,441.738,175.645,17.061,152.505
C08888=1093.425,51.876,441.722,175.647,17.062,152.505
C08889=1093.430,52.124,441.706,175.649,17.063,152.505
C08890=1093.435,52.374,441.690,175.651,17.065,152.505
C08891=1093.441,52.624,441.673,175.653,17.066,152.504
C08892=1093.447,52.873,441.657,175.655,17.067,152.504
C08893=1093.452,53.123,441.641,175.657,17.068,152.504
C08894=1093.458,53.372,441.626,175.660,17.070,152.504
C08895=1093.464,53.621,441.609,175.661,17.071,152.504
C08896=1093.470,53.870,441.593,175.664,17.072,152.504
C08897=1093.475,54.120,441.578,175.666,17.073,152.503
C08898=1093.481,54.370,441.561,175.667,17.074,152.503
C08899=1093.487,54.619,441.545,175.670,17.076,152.503
C08900=1093.493,54.868,441.529,175.672,17.076,152.503
C08901=1093.497,55.118,441.513,175.674,17.078,152.503
C08902=1093.503,55.367,441.497,175.676,17.079,152.503
C08903=1093.509,55.617,441.480,175.678,17.080,152.502
C08904=1093.515,55.866,441.464,175.680,17.082,152.502
C08905=1093.521,56.116,441.449,175.682,17.083,152.502
C08906=1093.527,56.365,441.432,175.684,17.084,152.502
C08907=1093.532,56.614,441.417,175.686,17.085,152.502
C08908=1093.538,56.863,441.400,175.689,17.086,152.502
C08909=1093.543,57.113,441.383,175.690,17.087,152.501
C08910=1093.549,57.362,441.367,175.693,17.089,152.501
C08911=1093.555,57.612,441.352,175.695,17.090,152.501
C08912=1093.561,57.862,441.335,175.697,17.091,152.501
C08913=1093.567,58.111,441.319,175.699,17.092,152.501
C08914=1093.573,58.360,441.303,175.701,17.094,152.501
C08915=1093.579,58.610,441.287,175.703,17.094,152.500
C08916=1093.584,58.859,441.270,175.705,17.096,152.500
C08917=1093.589,59.108,441.254,175.708,17.097,152.500
C08918=1093.595,59.357,441.238,175.709,17.098,152.500
C08919=1093.601,59.607,441.221,175.712,17.100,152.500
C08920=1093.607,59.856,441.205,175.714,17.100,152.499
C08921=1093.613,60.105,441.189,175.716,17.102,152.499
C08922=1093.618,60.356,441.173,175.718,17.103,152.499
C08923=1093.624,60.605,441.156,175.720,17.104,152.499
C08924=1093.630,60.854,441.140,175.722,17.105,152.499
C08925=1093.636,61.104,441.124,175.725,17.107,152.499
C08926=1093.642,61.353,441.108,175.727,17.107,152.498
C08927=1093.647,61.603,441.091,175.728,17.108,152.498
C08928=1093.653,61.852,441.075,175.731,17.110,152.498
C08929=1093.659,62.101,441.058,175.733,17.110,152.498
C08930=1093.665,62.351,441.042,175.735,17.112,152.498
C08931=1093.671,62.600,441.026,175.737,17.113,152.497
C08932=1093.676,62.849,441.008,175.740,17.114,152.497
C08933=1093.682,63.099,440.992,175.742,17.115,152.497
C08934=1093.689,63.374,440.974,175.744,17.117,152.497
C08935=1093.695,63.650,440.956,175.747,17.118,152.497
C08936=1093.702,63.925,440.938,175.749,17.118,152.496
C08937=1093.708,64.200,440.920,175.751,17.120,152.496
C08938=1093.714,64.450,440.904,175.754,17.121,152.496
C08939=1093.719,64.700,440.887,175.755,17.122,152.496
C08940=1093.725,64.949,440.871,175.758,17.124,152.496
C08941=1093.730,65.199,440.854,175.760,17.125,152.495
C08942=1093.736,65.448,440.837,175.762,17.126,152.495
C08943=1093.742,65.697,440.820,175.764,17.127,152.495
C08944=1093.748,65.946,440.804,175.767,17.128,152.495
C08945=1093.754,66.196,440.787,175.769,17.129,152.495
C08946=1093.759,66.445,440.770,175.770,17.130,152.494
C08947=1093.765,66.695,440.754,175.773,17.131,152.494
C08948=1093.771,66.944,440.738,175.775,17.132,152.494
C08949=1093.776,67.193,440.720,175.777,17.134,152.494
C08950=1093.782,67.442,440.704,175.779,17.135,152.494
C08951=1093.787,67.692,440.687,175.782,17.136,152.493
C08952=1093.793,67.941,440.671,175.783,17.137,152.493
C08953=1093.798,68.191,440.654,175.786,17.138,152.493
C08954=1093.805,68.440,440.637,175.788,17.139,152.493
C08955=1093.810,68.689,440.620,175.790,17.141,152.493
C08956=1093.816,68.939,440.604,175.792,17.141,152.492
C08957=1093.822,69.189,440.587,175.795,17.143,152.492
C08958=1093.828,69.438,440.570,175.797,17.144,152.492
C08959=1093.833,69.688,440.553,175.799,17.145,152.492
C08960=1093.839,69.937,440.537,175.801,17.146,152.492
C08961=1093.844,70.187,440.520,175.804,17.147,152.491
C08962=1093.851,70.435,440.503,175.806,17.148,152.491
C08963=1093.856,70.685,440.486,175.808,17.149,152.491
C08964=1093.862,70.934,440.470,175.810,17.150,152.491
C08965=1093.867,71.183,440.452,175.812,17.152,152.491
C08966=1093.872,71.433,440.435,175.814,17.152,152.490
C08967=1093.878,71.682,440.419,175.817,17.154,152.490
C08968=1093.884,71.931,440.402,175.819,17.155,152.490
C08969=1093.890,72.181,440.385,175.821,17.156,152.490
C08970=1093.895,72.430,440.369,175.823,17.157,152.490
C08971=1093.901,72.679,440.351,175.826,17.158,152.489
C08972=1093.907,72.929,440.335,175.828,17.159,152.489
C08973=1093.912,73.178,440.317,175.830,17.161,152.489
C08974=1093.919,73.428,440.300,175.832,17.161,152.489
C08975=1093.924,73.677,440.284,175.835,17.163,152.488
C08976=1093.929,73.927,440.266,175.836,17.163,152.488
C08977=1093.935,74.176,440.250,175.839,17.165,152.488
C08978=1093.941,74.425,440.232,175.841,17.166,152.488
C08979=1093.946,74.675,440.215,175.844,17.167,152.488
C08980=1093.952,74.924,440.199,175.845,17.168,152.488
C08981=1093.958,75.173,440.182,175.848,17.169,152.487
C08982=1093.963,75.423,440.165,175.850,17.170,152.487
C08983=1093.970,75.672,440.147,175.852,17.171,152.487
C08984=1093.975,75.922,440.131,175.854,17.172,152.487
C08985=1093.980,76.171,440.113,175.857,17.173,152.486
C08986=1093.986,76.420,440.097,175.859,17.174,152.486
C08987=1093.992,76.669,440.079,175.861,17.176,152.486
C08988=1093.997,76.919,440.062,175.863,17.176,152.486
C08989=1094.004,77.168,440.045,175.866,17.177,152.485
C08990=1094.009,77.418,440.028,175.868,17.178,152.485
C08991=1094.015,77.667,440.011,175.870,17.179,152.485
C08992=1094.020,77.916,439.993,175.873,17.181,152.485
C08993=1094.026,78.165,439.977,175.875,17.182,152.485
C08994=1094.032,78.414,439.959,175.877,17.183,152.484
C08995=1094.037,78.664,439.942,175.879,17.183,152.484
C08996=1094.043,78.914,439.924,175.882,17.185,152.484
C08997=1094.049,79.162,439.907,175.884,17.186,152.484
C08998=1094.055,79.439,439.889,175.886,17.187,152.483
C08999=1094.061,79.713,439.869,175.889,17.188,152.483
C09000=1094.067,79.989,439.850,175.891,17.189,152.483
C09001=1094.074,80.265,439.832,175.894,17.190,152.483
C09002=1094.079,80.514,439.814,175.896,17.192,152.482
C09003=1094.085,80.763,439.797,175.898,17.192,152.482
C09004=1094.090,81.013,439.780,175.901,17.194,152.482
C09005=1094.096,81.262,439.762,175.903,17.194,152.482
C09006=1094.102,81.511,439.744,175.905,17.196,152.482
C09007=1094.107,81.761,439.727,175.907,17.197,152.481
C09008=1094.112,82.010,439.710,175.910,17.198,152.481
C09009=1094.119,82.259,439.693,175.912,17.199,152.481
C09010=1094.124,82.509,439.676,175.914,17.200,152.481
C09011=1094.130,82.758,439.658,175.917,17.201,152.480
C09012=1094.135,83.007,439.640,175.919,17.202,152.480
C09013=1094.141,83.256,439.623,175.921,17.203,152.480
C09014=1094.146,83.506,439.606,175.923,17.204,152.480
C09015=1094.152,83.756,439.588,175.926,17.205,152.479
C09016=1094.158,84.005,439.571,175.928,17.206,152.479
C09017=1094.163,84.254,439.553,175.931,17.207,152.479
C09018=1094.169,84.503,439.536,175.933,17.208,152.479
C09019=1094.175,84.753,439.518,175.935,17.209,152.478
C09020=1094.180,85.002,439.501,175.937,17.209,152.478
C09021=1094.186,85.251,439.483,175.940,17.211,152.478
C09022=1094.191,85.500,439.465,175.942,17.212,152.478
C09023=1094.198,85.750,439.448,175.944,17.213,152.477
C09024=1094.203,85.999,439.431,175.947,17.214,152.477
C09025=1094.209,86.248,439.414,175.949,17.215,152.477
C09026=1094.215,86.498,439.396,175.952,17.216,152.477
C09027=1094.220,86.747,439.378,175.953,17.217,152.476
C09028=1094.226,86.996,439.361,175.956,17.218,152.476
C09029=1094.231,87.245,439.343,175.958,17.219,152.476
C09030=1094.238,87.495,439.325,175.961,17.220,152.476
C09031=1094.243,87.744,439.308,175.963,17.220,152.475
C09032=1094.249,87.993,439.290,175.965,17.222,152.475
C09033=1094.254,88.243,439.273,175.968,17.223,152.475
C09034=1094.260,88.492,439.255,175.970,17.224,152.475
C09035=1094.265,88.741,439.238,175.973,17.225,152.474
C09036=1094.272,88.991,439.220,175.975,17.225,152.474
C09037=1094.277,89.240,439.202,175.977,17.227,152.474
C09038=1094.283,89.489,439.185,175.979,17.227,152.474
C09039=1094.289,89.739,439.167,175.982,17.228,152.473
C09040=1094.294,89.988,439.149,175.984,17.229,152.473
C09041=1094.300,90.238,439.131,175.987,17.230,152.473
C09042=1094.306,90.487,439.114,175.989,17.232,152.472
C09043=1094.311,90.736,439.096,175.991,17.232,152.472
C09044=1094.318,90.986,439.078,175.994,17.233,152.472
C09045=1094.322,91.235,439.060,175.996,17.234,152.472
C09046=1094.328,91.484,439.042,175.999,17.235,152.471
C09047=1094.334,91.734,439.024,176.000,17.236,152.471
C09048=1094.339,91.983,439.007,176.003,17.237,152.471
C09049=1094.345,92.232,438.989,176.006,17.238,152.470
C09050=1094.351,92.481,438.970,176.008,17.239,152.470
C09051=1094.356,92.730,438.953,176.011,17.240,152.470
C09052=1094.362,92.979,438.935,176.013,17.240,152.470
C09053=1094.368,93.229,438.917,176.015,17.242,152.469
C09054=1094.373,93.478,438.899,176.017,17.242,152.469
C09055=1094.378,93.728,438.881,176.020,17.243,152.469
C09056=1094.384,93.977,438.863,176.023,17.245,152.469
C09057=1094.390,94.226,438.846,176.025,17.245,152.468
C09058=1094.396,94.476,438.828,176.027,17.247,152.468
C09059=1094.401,94.725,438.809,176.029,17.247,152.468
C09060=1094.406,94.974,438.791,176.032,17.248,152.468
C09061=1094.413,95.224,438.773,176.034,17.249,152.467
C09062=1094.419,95.499,438.754,176.037,17.250,152.467
C09063=1094.425,95.774,438.733,176.040,17.251,152.467
C09064=1094.431,96.050,438.714,176.042,17.252,152.466
C09065=1094.437,96.325,438.694,176.045,17.253,152.466
C09066=1094.443,96.575,438.676,176.047,17.254,152.466
C09067=1094.448,96.824,438.657,176.050,17.255,152.465
C09068=1094.454,97.074,438.639,176.053,17.256,152.465
C09069=1094.460,97.323,438.622,176.054,17.257,152.465
C09070=1094.466,97.572,438.604,176.057,17.258,152.465
C09071=1094.471,97.821,438.585,176.059,17.259,152.464
C09072=1094.477,98.070,438.567,176.062,17.259,152.464
C09073=1094.483,98.320,438.549,176.064,17.260,152.464
C09074=1094.488,98.569,438.531,176.067,17.261,152.463
C09075=1094.494,98.818,438.513,176.069,17.262,152.463
C09076=1094.500,99.067,438.495,176.072,17.263,152.463
C09077=1094.506,99.316,438.476,176.074,17.264,152.463
C09078=1094.511,99.566,438.458,176.076,17.264,152.462
C09079=1094.517,99.816,438.440,176.079,17.266,152.462
C09080=1094.523,100.064,438.422,176.082,17.266,152.462
C09081=1094.528,100.314,438.404,176.084,17.267,152.461
C09082=1094.534,100.563,438.386,176.087,17.268,152.461
C09083=1094.540,100.812,438.367,176.088,17.269,152.461
C09084=1094.545,101.062,438.349,176.091,17.270,152.460
C09085=1094.551,101.311,438.330,176.094,17.271,152.460
C09086=1094.556,101.560,438.312,176.096,17.271,152.460
C09087=1094.562,101.810,438.294,176.099,17.273,152.460
C09088=1094.567,102.058,438.276,176.101,17.273,152.459
C09089=1094.573,102.308,438.258,176.104,17.274,152.459
C09090=1094.578,102.557,438.239,176.106,17.275,152.459
C09091=1094.585,102.807,438.221,176.108,17.276,152.458
